Fanuc TP program (LS listing): hosenrohr_ov_h802.ls

/PROG  hosenrohr_ov_h802
/ATTR
COMMENT	= "19-02-26 08:34:14";
PROG_SIZE	= 0;
DEFAULT_GROUP	= 1, 1, *, *, *;
/APPL
    ARC Welding Equipment: 1, *, *, *, *;
/MN
   1:  CALL HOME_ALL;
   1:  UFRAME_NUM = 1;
   1:  UTOOL_NUM = 3;
   1:  COL GUARD ADJUST 150;
   1:  ! -- Layer/Ebene 72 -- !;
   1:  PR[91] = PR[90];
   1:  PR[GP1:91,1] = PR[GP1:90,1] + -1.017;
   1:  PR[GP1:91,2] = PR[GP1:90,2] + 18.874;
   1:  PR[GP1:91,3] = PR[GP1:90,3] + 44.225;
   1:  !Sicherheitspunkt!;
   1:  PR[92] = PR[91];
   1:  PR[92] = PR[GP1:92,3] + 50;
   1:J PR[92];
   1:  !Schweissanfang anfahren!;
   1:L PR[91] R[100]mm/sec CNT100;
   1:  CALL LASER_DRAHT_START;
   1:  PR[GP1:91,1] = PR[GP1:90,1] + -3.858;
   1:  PR[GP1:91,2] = PR[GP1:90,2] + 20.009;
   1:L PR[91] R[100]mm/sec CNT100;
   1:  PR[GP1:91,1] = PR[GP1:90,1] + -5.422;
   1:  PR[GP1:91,2] = PR[GP1:90,2] + 20.569;
   1:L PR[91] R[100]mm/sec CNT100;
   1:  PR[GP1:91,1] = PR[GP1:90,1] + -10.694;
   1:  PR[GP1:91,2] = PR[GP1:90,2] + 21.232;
   1:L PR[91] R[100]mm/sec CNT100;
   1:  PR[GP1:91,1] = PR[GP1:90,1] + -11.339;
   1:  PR[GP1:91,2] = PR[GP1:90,2] + 21.294;
   1:L PR[91] R[100]mm/sec CNT100;
   1:  PR[GP1:91,1] = PR[GP1:90,1] + -17.031;
   1:  PR[GP1:91,2] = PR[GP1:90,2] + 20.547;
   1:L PR[91] R[100]mm/sec CNT100;
   1:  PR[GP1:91,1] = PR[GP1:90,1] + -17.231;
   1:  PR[GP1:91,2] = PR[GP1:90,2] + 20.514;
   1:L PR[91] R[100]mm/sec CNT100;
   1:  PR[GP1:91,1] = PR[GP1:90,1] + -22.722;
   1:  PR[GP1:91,2] = PR[GP1:90,2] + 18.298;
   1:L PR[91] R[100]mm/sec CNT100;
   1:  PR[GP1:91,1] = PR[GP1:90,1] + -27.488;
   1:  PR[GP1:91,2] = PR[GP1:90,2] + 14.829;
   1:L PR[91] R[100]mm/sec CNT100;
   1:  PR[GP1:91,1] = PR[GP1:90,1] + -27.511;
   1:  PR[GP1:91,2] = PR[GP1:90,2] + 14.804;
   1:L PR[91] R[100]mm/sec CNT100;
   1:  PR[GP1:91,1] = PR[GP1:90,1] + -30.986;
   1:  PR[GP1:91,2] = PR[GP1:90,2] + 10.489;
   1:L PR[91] R[100]mm/sec CNT100;
   1:  PR[GP1:91,1] = PR[GP1:90,1] + -31.085;
   1:  PR[GP1:91,2] = PR[GP1:90,2] + 10.338;
   1:L PR[91] R[100]mm/sec CNT100;
   1:  PR[GP1:91,1] = PR[GP1:90,1] + -33.300;
   1:  PR[GP1:91,2] = PR[GP1:90,2] + 5.293;
   1:L PR[91] R[100]mm/sec CNT100;
   1:  PR[GP1:91,1] = PR[GP1:90,1] + -33.354;
   1:  PR[GP1:91,2] = PR[GP1:90,2] + 5.083;
   1:L PR[91] R[100]mm/sec CNT100;
   1:  PR[GP1:91,1] = PR[GP1:90,1] + -33.385;
   1:  PR[GP1:91,2] = PR[GP1:90,2] + 4.702;
   1:L PR[91] R[100]mm/sec CNT100;
   1:  PR[GP1:91,1] = PR[GP1:90,1] + -34.086;
   1:  PR[GP1:91,2] = PR[GP1:90,2] + -0.354;
   1:L PR[91] R[100]mm/sec CNT100;
   1:  PR[GP1:91,1] = PR[GP1:90,1] + -34.060;
   1:  PR[GP1:91,2] = PR[GP1:90,2] + -0.674;
   1:L PR[91] R[100]mm/sec CNT100;
   1:  PR[GP1:91,1] = PR[GP1:90,1] + -33.363;
   1:  PR[GP1:91,2] = PR[GP1:90,2] + -5.673;
   1:L PR[91] R[100]mm/sec CNT100;
   1:  PR[GP1:91,1] = PR[GP1:90,1] + -33.300;
   1:  PR[GP1:91,2] = PR[GP1:90,2] + -5.917;
   1:L PR[91] R[100]mm/sec CNT100;
   1:  PR[GP1:91,1] = PR[GP1:90,1] + -33.156;
   1:  PR[GP1:91,2] = PR[GP1:90,2] + -6.238;
   1:L PR[91] R[100]mm/sec CNT100;
   1:  PR[GP1:91,1] = PR[GP1:90,1] + -31.078;
   1:  PR[GP1:91,2] = PR[GP1:90,2] + -10.975;
   1:L PR[91] R[100]mm/sec CNT100;
   1:  PR[GP1:91,1] = PR[GP1:90,1] + -30.980;
   1:  PR[GP1:91,2] = PR[GP1:90,2] + -11.125;
   1:L PR[91] R[100]mm/sec CNT100;
   1:  PR[GP1:91,1] = PR[GP1:90,1] + -27.495;
   1:  PR[GP1:91,2] = PR[GP1:90,2] + -15.443;
   1:L PR[91] R[100]mm/sec CNT100;
   1:  PR[GP1:91,1] = PR[GP1:90,1] + -27.473;
   1:  PR[GP1:91,2] = PR[GP1:90,2] + -15.467;
   1:L PR[91] R[100]mm/sec CNT100;
   1:  PR[GP1:91,1] = PR[GP1:90,1] + -22.696;
   1:  PR[GP1:91,2] = PR[GP1:90,2] + -18.937;
   1:L PR[91] R[100]mm/sec CNT100;
   1:  PR[GP1:91,1] = PR[GP1:90,1] + -17.195;
   1:  PR[GP1:91,2] = PR[GP1:90,2] + -21.148;
   1:L PR[91] R[100]mm/sec CNT100;
   1:  PR[GP1:91,1] = PR[GP1:90,1] + -16.992;
   1:  PR[GP1:91,2] = PR[GP1:90,2] + -21.180;
   1:L PR[91] R[100]mm/sec CNT100;
   1:  PR[GP1:91,1] = PR[GP1:90,1] + -11.296;
   1:  PR[GP1:91,2] = PR[GP1:90,2] + -21.918;
   1:L PR[91] R[100]mm/sec CNT100;
   1:  PR[GP1:91,1] = PR[GP1:90,1] + -10.640;
   1:  PR[GP1:91,2] = PR[GP1:90,2] + -21.853;
   1:L PR[91] R[100]mm/sec CNT100;
   1:  PR[GP1:91,1] = PR[GP1:90,1] + -5.365;
   1:  PR[GP1:91,2] = PR[GP1:90,2] + -21.179;
   1:L PR[91] R[100]mm/sec CNT100;
   1:  PR[GP1:91,1] = PR[GP1:90,1] + -4.473;
   1:  PR[GP1:91,2] = PR[GP1:90,2] + -20.868;
   1:L PR[91] R[100]mm/sec CNT100;
   1:  PR[GP1:91,1] = PR[GP1:90,1] + -1.022;
   1:  PR[GP1:91,2] = PR[GP1:90,2] + -19.515;
   1:L PR[91] R[100]mm/sec CNT100;
   1:  PR[GP1:91,1] = PR[GP1:90,1] + 0.411;
   1:  PR[GP1:91,2] = PR[GP1:90,2] + -19.282;
   1:L PR[91] R[100]mm/sec CNT100;
   1:  PR[GP1:91,1] = PR[GP1:90,1] + 1.272;
   1:  PR[GP1:91,2] = PR[GP1:90,2] + -19.552;
   1:L PR[91] R[100]mm/sec CNT100;
   1:  PR[GP1:91,1] = PR[GP1:90,1] + 4.630;
   1:  PR[GP1:91,2] = PR[GP1:90,2] + -20.867;
   1:L PR[91] R[100]mm/sec CNT100;
   1:  PR[GP1:91,1] = PR[GP1:90,1] + 5.411;
   1:  PR[GP1:91,2] = PR[GP1:90,2] + -21.143;
   1:L PR[91] R[100]mm/sec CNT100;
   1:  PR[GP1:91,1] = PR[GP1:90,1] + 10.700;
   1:  PR[GP1:91,2] = PR[GP1:90,2] + -21.827;
   1:L PR[91] R[100]mm/sec CNT100;
   1:  PR[GP1:91,1] = PR[GP1:90,1] + 10.853;
   1:  PR[GP1:91,2] = PR[GP1:90,2] + -21.859;
   1:L PR[91] R[100]mm/sec CNT100;
   1:  PR[GP1:91,1] = PR[GP1:90,1] + 11.450;
   1:  PR[GP1:91,2] = PR[GP1:90,2] + -21.918;
   1:L PR[91] R[100]mm/sec CNT100;
   1:  PR[GP1:91,1] = PR[GP1:90,1] + 17.146;
   1:  PR[GP1:91,2] = PR[GP1:90,2] + -21.180;
   1:L PR[91] R[100]mm/sec CNT100;
   1:  PR[GP1:91,1] = PR[GP1:90,1] + 17.349;
   1:  PR[GP1:91,2] = PR[GP1:90,2] + -21.148;
   1:L PR[91] R[100]mm/sec CNT100;
   1:  PR[GP1:91,1] = PR[GP1:90,1] + 22.851;
   1:  PR[GP1:91,2] = PR[GP1:90,2] + -18.939;
   1:L PR[91] R[100]mm/sec CNT100;
   1:  PR[GP1:91,1] = PR[GP1:90,1] + 27.626;
   1:  PR[GP1:91,2] = PR[GP1:90,2] + -15.472;
   1:L PR[91] R[100]mm/sec CNT100;
   1:  PR[GP1:91,1] = PR[GP1:90,1] + 27.648;
   1:  PR[GP1:91,2] = PR[GP1:90,2] + -15.448;
   1:L PR[91] R[100]mm/sec CNT100;
   1:  PR[GP1:91,1] = PR[GP1:90,1] + 31.132;
   1:  PR[GP1:91,2] = PR[GP1:90,2] + -11.122;
   1:L PR[91] R[100]mm/sec CNT100;
   1:  PR[GP1:91,1] = PR[GP1:90,1] + 31.234;
   1:  PR[GP1:91,2] = PR[GP1:90,2] + -10.967;
   1:L PR[91] R[100]mm/sec CNT100;
   1:  PR[GP1:91,1] = PR[GP1:90,1] + 33.454;
   1:  PR[GP1:91,2] = PR[GP1:90,2] + -5.943;
   1:L PR[91] R[100]mm/sec CNT100;
   1:  PR[GP1:91,1] = PR[GP1:90,1] + 33.508;
   1:  PR[GP1:91,2] = PR[GP1:90,2] + -5.738;
   1:L PR[91] R[100]mm/sec CNT100;
   1:  PR[GP1:91,1] = PR[GP1:90,1] + 33.540;
   1:  PR[GP1:91,2] = PR[GP1:90,2] + -5.345;
   1:L PR[91] R[100]mm/sec CNT100;
   1:  PR[GP1:91,1] = PR[GP1:90,1] + 34.242;
   1:  PR[GP1:91,2] = PR[GP1:90,2] + -0.271;
   1:L PR[91] R[100]mm/sec CNT100;
   1:  PR[GP1:91,1] = PR[GP1:90,1] + 34.215;
   1:  PR[GP1:91,2] = PR[GP1:90,2] + 0.065;
   1:L PR[91] R[100]mm/sec CNT100;
   1:  PR[GP1:91,1] = PR[GP1:90,1] + 33.520;
   1:  PR[GP1:91,2] = PR[GP1:90,2] + 5.069;
   1:L PR[91] R[100]mm/sec CNT100;
   1:  PR[GP1:91,1] = PR[GP1:90,1] + 33.456;
   1:  PR[GP1:91,2] = PR[GP1:90,2] + 5.313;
   1:L PR[91] R[100]mm/sec CNT100;
   1:  PR[GP1:91,1] = PR[GP1:90,1] + 31.241;
   1:  PR[GP1:91,2] = PR[GP1:90,2] + 10.332;
   1:L PR[91] R[100]mm/sec CNT100;
   1:  PR[GP1:91,1] = PR[GP1:90,1] + 31.139;
   1:  PR[GP1:91,2] = PR[GP1:90,2] + 10.487;
   1:L PR[91] R[100]mm/sec CNT100;
   1:  PR[GP1:91,1] = PR[GP1:90,1] + 27.664;
   1:  PR[GP1:91,2] = PR[GP1:90,2] + 14.809;
   1:L PR[91] R[100]mm/sec CNT100;
   1:  PR[GP1:91,1] = PR[GP1:90,1] + 27.641;
   1:  PR[GP1:91,2] = PR[GP1:90,2] + 14.834;
   1:L PR[91] R[100]mm/sec CNT100;
   1:  PR[GP1:91,1] = PR[GP1:90,1] + 22.877;
   1:  PR[GP1:91,2] = PR[GP1:90,2] + 18.301;
   1:L PR[91] R[100]mm/sec CNT100;
   1:  PR[GP1:91,1] = PR[GP1:90,1] + 17.385;
   1:  PR[GP1:91,2] = PR[GP1:90,2] + 20.514;
   1:L PR[91] R[100]mm/sec CNT100;
   1:  PR[GP1:91,1] = PR[GP1:90,1] + 17.184;
   1:  PR[GP1:91,2] = PR[GP1:90,2] + 20.547;
   1:L PR[91] R[100]mm/sec CNT100;
   1:  PR[GP1:91,1] = PR[GP1:90,1] + 11.493;
   1:  PR[GP1:91,2] = PR[GP1:90,2] + 21.294;
   1:L PR[91] R[100]mm/sec CNT100;
   1:  PR[GP1:91,1] = PR[GP1:90,1] + 10.848;
   1:  PR[GP1:91,2] = PR[GP1:90,2] + 21.232;
   1:L PR[91] R[100]mm/sec CNT100;
   1:  PR[GP1:91,1] = PR[GP1:90,1] + 5.555;
   1:  PR[GP1:91,2] = PR[GP1:90,2] + 20.565;
   1:L PR[91] R[100]mm/sec CNT100;
   1:  PR[GP1:91,1] = PR[GP1:90,1] + 5.340;
   1:  PR[GP1:91,2] = PR[GP1:90,2] + 20.494;
   1:L PR[91] R[100]mm/sec CNT100;
   1:  PR[GP1:91,1] = PR[GP1:90,1] + 4.017;
   1:  PR[GP1:91,2] = PR[GP1:90,2] + 20.009;
   1:L PR[91] R[100]mm/sec CNT100;
   1:  PR[GP1:91,1] = PR[GP1:90,1] + 1.242;
   1:  PR[GP1:91,2] = PR[GP1:90,2] + 18.902;
   1:L PR[91] R[100]mm/sec CNT100;
   1:  PR[GP1:91,1] = PR[GP1:90,1] + 0.855;
   1:  PR[GP1:91,2] = PR[GP1:90,2] + 18.802;
   1:L PR[91] R[100]mm/sec CNT100;
   1:  PR[GP1:91,1] = PR[GP1:90,1] + 0.519;
   1:  PR[GP1:91,2] = PR[GP1:90,2] + 18.647;
   1:L PR[91] R[100]mm/sec CNT100;
   1:  ! -- Layer/Ebene 73 -- !;
   1:  PR[91] = PR[90];
   1:  PR[GP1:91,1] = PR[GP1:90,1] + -1.002;
   1:  PR[GP1:91,2] = PR[GP1:90,2] + 19.074;
   1:  PR[GP1:91,3] = PR[GP1:90,3] + 44.835;
   1:L PR[91] R[100]mm/sec CNT100;
   1:  PR[GP1:91,1] = PR[GP1:90,1] + -3.287;
   1:  PR[GP1:91,2] = PR[GP1:90,2] + 19.987;
   1:L PR[91] R[100]mm/sec CNT100;
   1:  PR[GP1:91,1] = PR[GP1:90,1] + -5.044;
   1:  PR[GP1:91,2] = PR[GP1:90,2] + 20.628;
   1:L PR[91] R[100]mm/sec CNT100;
   1:  PR[GP1:91,1] = PR[GP1:90,1] + -5.181;
   1:  PR[GP1:91,2] = PR[GP1:90,2] + 20.671;
   1:L PR[91] R[100]mm/sec CNT100;
   1:  PR[GP1:91,1] = PR[GP1:90,1] + -10.231;
   1:  PR[GP1:91,2] = PR[GP1:90,2] + 21.306;
   1:L PR[91] R[100]mm/sec CNT100;
   1:  PR[GP1:91,1] = PR[GP1:90,1] + -11.140;
   1:  PR[GP1:91,2] = PR[GP1:90,2] + 21.393;
   1:L PR[91] R[100]mm/sec CNT100;
   1:  PR[GP1:91,1] = PR[GP1:90,1] + -16.581;
   1:  PR[GP1:91,2] = PR[GP1:90,2] + 20.679;
   1:L PR[91] R[100]mm/sec CNT100;
   1:  PR[GP1:91,1] = PR[GP1:90,1] + -17.045;
   1:  PR[GP1:91,2] = PR[GP1:90,2] + 20.605;
   1:L PR[91] R[100]mm/sec CNT100;
   1:  PR[GP1:91,1] = PR[GP1:90,1] + -22.543;
   1:  PR[GP1:91,2] = PR[GP1:90,2] + 18.372;
   1:L PR[91] R[100]mm/sec CNT100;
   1:  PR[GP1:91,1] = PR[GP1:90,1] + -25.480;
   1:  PR[GP1:91,2] = PR[GP1:90,2] + 16.189;
   1:L PR[91] R[100]mm/sec CNT100;
   1:  PR[GP1:91,1] = PR[GP1:90,1] + -27.252;
   1:  PR[GP1:91,2] = PR[GP1:90,2] + 14.898;
   1:L PR[91] R[100]mm/sec CNT100;
   1:  PR[GP1:91,1] = PR[GP1:90,1] + -30.851;
   1:  PR[GP1:91,2] = PR[GP1:90,2] + 10.438;
   1:L PR[91] R[100]mm/sec CNT100;
   1:  PR[GP1:91,1] = PR[GP1:90,1] + -30.874;
   1:  PR[GP1:91,2] = PR[GP1:90,2] + 10.403;
   1:L PR[91] R[100]mm/sec CNT100;
   1:  PR[GP1:91,1] = PR[GP1:90,1] + -30.924;
   1:  PR[GP1:91,2] = PR[GP1:90,2] + 10.292;
   1:L PR[91] R[100]mm/sec CNT100;
   1:  PR[GP1:91,1] = PR[GP1:90,1] + -33.125;
   1:  PR[GP1:91,2] = PR[GP1:90,2] + 5.268;
   1:L PR[91] R[100]mm/sec CNT100;
   1:  PR[GP1:91,1] = PR[GP1:90,1] + -33.144;
   1:  PR[GP1:91,2] = PR[GP1:90,2] + 5.195;
   1:L PR[91] R[100]mm/sec CNT100;
   1:  PR[GP1:91,1] = PR[GP1:90,1] + -33.163;
   1:  PR[GP1:91,2] = PR[GP1:90,2] + 4.957;
   1:L PR[91] R[100]mm/sec CNT100;
   1:  PR[GP1:91,1] = PR[GP1:90,1] + -33.900;
   1:  PR[GP1:91,2] = PR[GP1:90,2] + -0.354;
   1:L PR[91] R[100]mm/sec CNT100;
   1:  PR[GP1:91,1] = PR[GP1:90,1] + -33.885;
   1:  PR[GP1:91,2] = PR[GP1:90,2] + -0.535;
   1:L PR[91] R[100]mm/sec CNT100;
   1:  PR[GP1:91,1] = PR[GP1:90,1] + -33.153;
   1:  PR[GP1:91,2] = PR[GP1:90,2] + -5.784;
   1:L PR[91] R[100]mm/sec CNT100;
   1:  PR[GP1:91,1] = PR[GP1:90,1] + -33.125;
   1:  PR[GP1:91,2] = PR[GP1:90,2] + -5.892;
   1:L PR[91] R[100]mm/sec CNT100;
   1:  PR[GP1:91,1] = PR[GP1:90,1] + -33.040;
   1:  PR[GP1:91,2] = PR[GP1:90,2] + -6.081;
   1:L PR[91] R[100]mm/sec CNT100;
   1:  PR[GP1:91,1] = PR[GP1:90,1] + -30.863;
   1:  PR[GP1:91,2] = PR[GP1:90,2] + -11.044;
   1:L PR[91] R[100]mm/sec CNT100;
   1:  PR[GP1:91,1] = PR[GP1:90,1] + -30.844;
   1:  PR[GP1:91,2] = PR[GP1:90,2] + -11.074;
   1:L PR[91] R[100]mm/sec CNT100;
   1:  PR[GP1:91,1] = PR[GP1:90,1] + -27.236;
   1:  PR[GP1:91,2] = PR[GP1:90,2] + -15.537;
   1:L PR[91] R[100]mm/sec CNT100;
   1:  PR[GP1:91,1] = PR[GP1:90,1] + -25.483;
   1:  PR[GP1:91,2] = PR[GP1:90,2] + -16.812;
   1:L PR[91] R[100]mm/sec CNT100;
   1:  PR[GP1:91,1] = PR[GP1:90,1] + -22.517;
   1:  PR[GP1:91,2] = PR[GP1:90,2] + -19.010;
   1:L PR[91] R[100]mm/sec CNT100;
   1:  PR[GP1:91,1] = PR[GP1:90,1] + -17.009;
   1:  PR[GP1:91,2] = PR[GP1:90,2] + -21.238;
   1:L PR[91] R[100]mm/sec CNT100;
   1:  PR[GP1:91,1] = PR[GP1:90,1] + -16.542;
   1:  PR[GP1:91,2] = PR[GP1:90,2] + -21.312;
   1:L PR[91] R[100]mm/sec CNT100;
   1:  PR[GP1:91,1] = PR[GP1:90,1] + -11.097;
   1:  PR[GP1:91,2] = PR[GP1:90,2] + -22.018;
   1:L PR[91] R[100]mm/sec CNT100;
   1:  PR[GP1:91,1] = PR[GP1:90,1] + -10.175;
   1:  PR[GP1:91,2] = PR[GP1:90,2] + -21.926;
   1:L PR[91] R[100]mm/sec CNT100;
   1:  PR[GP1:91,1] = PR[GP1:90,1] + -5.149;
   1:  PR[GP1:91,2] = PR[GP1:90,2] + -21.284;
   1:L PR[91] R[100]mm/sec CNT100;
   1:  PR[GP1:91,1] = PR[GP1:90,1] + -4.038;
   1:  PR[GP1:91,2] = PR[GP1:90,2] + -20.897;
   1:L PR[91] R[100]mm/sec CNT100;
   1:  PR[GP1:91,1] = PR[GP1:90,1] + -1.002;
   1:  PR[GP1:91,2] = PR[GP1:90,2] + -19.707;
   1:L PR[91] R[100]mm/sec CNT100;
   1:  PR[GP1:91,1] = PR[GP1:90,1] + 0.577;
   1:  PR[GP1:91,2] = PR[GP1:90,2] + -19.458;
   1:L PR[91] R[100]mm/sec CNT100;
   1:  PR[GP1:91,1] = PR[GP1:90,1] + 0.929;
   1:  PR[GP1:91,2] = PR[GP1:90,2] + -19.646;
   1:L PR[91] R[100]mm/sec CNT100;
   1:  PR[GP1:91,1] = PR[GP1:90,1] + 1.247;
   1:  PR[GP1:91,2] = PR[GP1:90,2] + -19.742;
   1:L PR[91] R[100]mm/sec CNT100;
   1:  PR[GP1:91,1] = PR[GP1:90,1] + 4.196;
   1:  PR[GP1:91,2] = PR[GP1:90,2] + -20.896;
   1:L PR[91] R[100]mm/sec CNT100;
   1:  PR[GP1:91,1] = PR[GP1:90,1] + 5.172;
   1:  PR[GP1:91,2] = PR[GP1:90,2] + -21.240;
   1:L PR[91] R[100]mm/sec CNT100;
   1:  PR[GP1:91,1] = PR[GP1:90,1] + 10.180;
   1:  PR[GP1:91,2] = PR[GP1:90,2] + -21.888;
   1:L PR[91] R[100]mm/sec CNT100;
   1:  PR[GP1:91,1] = PR[GP1:90,1] + 10.388;
   1:  PR[GP1:91,2] = PR[GP1:90,2] + -21.932;
   1:L PR[91] R[100]mm/sec CNT100;
   1:  PR[GP1:91,1] = PR[GP1:90,1] + 11.251;
   1:  PR[GP1:91,2] = PR[GP1:90,2] + -22.018;
   1:L PR[91] R[100]mm/sec CNT100;
   1:  PR[GP1:91,1] = PR[GP1:90,1] + 16.697;
   1:  PR[GP1:91,2] = PR[GP1:90,2] + -21.312;
   1:L PR[91] R[100]mm/sec CNT100;
   1:  PR[GP1:91,1] = PR[GP1:90,1] + 17.164;
   1:  PR[GP1:91,2] = PR[GP1:90,2] + -21.238;
   1:L PR[91] R[100]mm/sec CNT100;
   1:  PR[GP1:91,1] = PR[GP1:90,1] + 22.673;
   1:  PR[GP1:91,2] = PR[GP1:90,2] + -19.012;
   1:L PR[91] R[100]mm/sec CNT100;
   1:  PR[GP1:91,1] = PR[GP1:90,1] + 25.638;
   1:  PR[GP1:91,2] = PR[GP1:90,2] + -16.814;
   1:L PR[91] R[100]mm/sec CNT100;
   1:  PR[GP1:91,1] = PR[GP1:90,1] + 27.390;
   1:  PR[GP1:91,2] = PR[GP1:90,2] + -15.541;
   1:L PR[91] R[100]mm/sec CNT100;
   1:  PR[GP1:91,1] = PR[GP1:90,1] + 30.998;
   1:  PR[GP1:91,2] = PR[GP1:90,2] + -11.069;
   1:L PR[91] R[100]mm/sec CNT100;
   1:  PR[GP1:91,1] = PR[GP1:90,1] + 31.020;
   1:  PR[GP1:91,2] = PR[GP1:90,2] + -11.036;
   1:L PR[91] R[100]mm/sec CNT100;
   1:  PR[GP1:91,1] = PR[GP1:90,1] + 33.280;
   1:  PR[GP1:91,2] = PR[GP1:90,2] + -5.916;
   1:L PR[91] R[100]mm/sec CNT100;
   1:  PR[GP1:91,1] = PR[GP1:90,1] + 33.298;
   1:  PR[GP1:91,2] = PR[GP1:90,2] + -5.846;
   1:L PR[91] R[100]mm/sec CNT100;
   1:  PR[GP1:91,1] = PR[GP1:90,1] + 33.318;
   1:  PR[GP1:91,2] = PR[GP1:90,2] + -5.601;
   1:L PR[91] R[100]mm/sec CNT100;
   1:  PR[GP1:91,1] = PR[GP1:90,1] + 34.056;
   1:  PR[GP1:91,2] = PR[GP1:90,2] + -0.271;
   1:L PR[91] R[100]mm/sec CNT100;
   1:  PR[GP1:91,1] = PR[GP1:90,1] + 34.040;
   1:  PR[GP1:91,2] = PR[GP1:90,2] + -0.079;
   1:L PR[91] R[100]mm/sec CNT100;
   1:  PR[GP1:91,1] = PR[GP1:90,1] + 33.310;
   1:  PR[GP1:91,2] = PR[GP1:90,2] + 5.176;
   1:L PR[91] R[100]mm/sec CNT100;
   1:  PR[GP1:91,1] = PR[GP1:90,1] + 33.282;
   1:  PR[GP1:91,2] = PR[GP1:90,2] + 5.286;
   1:L PR[91] R[100]mm/sec CNT100;
   1:  PR[GP1:91,1] = PR[GP1:90,1] + 31.027;
   1:  PR[GP1:91,2] = PR[GP1:90,2] + 10.400;
   1:L PR[91] R[100]mm/sec CNT100;
   1:  PR[GP1:91,1] = PR[GP1:90,1] + 31.005;
   1:  PR[GP1:91,2] = PR[GP1:90,2] + 10.433;
   1:L PR[91] R[100]mm/sec CNT100;
   1:  PR[GP1:91,1] = PR[GP1:90,1] + 27.406;
   1:  PR[GP1:91,2] = PR[GP1:90,2] + 14.902;
   1:L PR[91] R[100]mm/sec CNT100;
   1:  PR[GP1:91,1] = PR[GP1:90,1] + 25.636;
   1:  PR[GP1:91,2] = PR[GP1:90,2] + 16.190;
   1:L PR[91] R[100]mm/sec CNT100;
   1:  PR[GP1:91,1] = PR[GP1:90,1] + 22.698;
   1:  PR[GP1:91,2] = PR[GP1:90,2] + 18.374;
   1:L PR[91] R[100]mm/sec CNT100;
   1:  PR[GP1:91,1] = PR[GP1:90,1] + 17.199;
   1:  PR[GP1:91,2] = PR[GP1:90,2] + 20.605;
   1:L PR[91] R[100]mm/sec CNT100;
   1:  PR[GP1:91,1] = PR[GP1:90,1] + 16.735;
   1:  PR[GP1:91,2] = PR[GP1:90,2] + 20.679;
   1:L PR[91] R[100]mm/sec CNT100;
   1:  PR[GP1:91,1] = PR[GP1:90,1] + 11.294;
   1:  PR[GP1:91,2] = PR[GP1:90,2] + 21.394;
   1:L PR[91] R[100]mm/sec CNT100;
   1:  PR[GP1:91,1] = PR[GP1:90,1] + 10.386;
   1:  PR[GP1:91,2] = PR[GP1:90,2] + 21.306;
   1:L PR[91] R[100]mm/sec CNT100;
   1:  PR[GP1:91,1] = PR[GP1:90,1] + 5.339;
   1:  PR[GP1:91,2] = PR[GP1:90,2] + 20.670;
   1:L PR[91] R[100]mm/sec CNT100;
   1:  PR[GP1:91,1] = PR[GP1:90,1] + 5.047;
   1:  PR[GP1:91,2] = PR[GP1:90,2] + 20.575;
   1:L PR[91] R[100]mm/sec CNT100;
   1:  PR[GP1:91,1] = PR[GP1:90,1] + 3.442;
   1:  PR[GP1:91,2] = PR[GP1:90,2] + 19.986;
   1:L PR[91] R[100]mm/sec CNT100;
   1:  PR[GP1:91,1] = PR[GP1:90,1] + 1.226;
   1:  PR[GP1:91,2] = PR[GP1:90,2] + 19.101;
   1:L PR[91] R[100]mm/sec CNT100;
   1:  PR[GP1:91,1] = PR[GP1:90,1] + 0.926;
   1:  PR[GP1:91,2] = PR[GP1:90,2] + 19.024;
   1:L PR[91] R[100]mm/sec CNT100;
   1:  PR[GP1:91,1] = PR[GP1:90,1] + 0.534;
   1:  PR[GP1:91,2] = PR[GP1:90,2] + 18.843;
   1:L PR[91] R[100]mm/sec CNT100;
   1:  ! -- Layer/Ebene 74 -- !;
   1:  PR[91] = PR[90];
   1:  PR[GP1:91,1] = PR[GP1:90,1] + -0.986;
   1:  PR[GP1:91,2] = PR[GP1:90,2] + 19.274;
   1:  PR[GP1:91,3] = PR[GP1:90,3] + 45.445;
   1:L PR[91] R[100]mm/sec CNT100;
   1:  PR[GP1:91,1] = PR[GP1:90,1] + -2.711;
   1:  PR[GP1:91,2] = PR[GP1:90,2] + 19.963;
   1:L PR[91] R[100]mm/sec CNT100;
   1:  PR[GP1:91,1] = PR[GP1:90,1] + -4.778;
   1:  PR[GP1:91,2] = PR[GP1:90,2] + 20.717;
   1:L PR[91] R[100]mm/sec CNT100;
   1:  PR[GP1:91,1] = PR[GP1:90,1] + -4.964;
   1:  PR[GP1:91,2] = PR[GP1:90,2] + 20.776;
   1:L PR[91] R[100]mm/sec CNT100;
   1:  PR[GP1:91,1] = PR[GP1:90,1] + -9.769;
   1:  PR[GP1:91,2] = PR[GP1:90,2] + 21.380;
   1:L PR[91] R[100]mm/sec CNT100;
   1:  PR[GP1:91,1] = PR[GP1:90,1] + -10.941;
   1:  PR[GP1:91,2] = PR[GP1:90,2] + 21.493;
   1:L PR[91] R[100]mm/sec CNT100;
   1:  PR[GP1:91,1] = PR[GP1:90,1] + -16.132;
   1:  PR[GP1:91,2] = PR[GP1:90,2] + 20.811;
   1:L PR[91] R[100]mm/sec CNT100;
   1:  PR[GP1:91,1] = PR[GP1:90,1] + -16.861;
   1:  PR[GP1:91,2] = PR[GP1:90,2] + 20.695;
   1:L PR[91] R[100]mm/sec CNT100;
   1:  PR[GP1:91,1] = PR[GP1:90,1] + -22.059;
   1:  PR[GP1:91,2] = PR[GP1:90,2] + 18.590;
   1:L PR[91] R[100]mm/sec CNT100;
   1:  PR[GP1:91,1] = PR[GP1:90,1] + -22.355;
   1:  PR[GP1:91,2] = PR[GP1:90,2] + 18.460;
   1:L PR[91] R[100]mm/sec CNT100;
   1:  PR[GP1:91,1] = PR[GP1:90,1] + -27.062;
   1:  PR[GP1:91,2] = PR[GP1:90,2] + 14.958;
   1:L PR[91] R[100]mm/sec CNT100;
   1:  PR[GP1:91,1] = PR[GP1:90,1] + -28.678;
   1:  PR[GP1:91,2] = PR[GP1:90,2] + 12.917;
   1:L PR[91] R[100]mm/sec CNT100;
   1:  PR[GP1:91,1] = PR[GP1:90,1] + -30.671;
   1:  PR[GP1:91,2] = PR[GP1:90,2] + 10.441;
   1:L PR[91] R[100]mm/sec CNT100;
   1:  PR[GP1:91,1] = PR[GP1:90,1] + -32.946;
   1:  PR[GP1:91,2] = PR[GP1:90,2] + 5.252;
   1:L PR[91] R[100]mm/sec CNT100;
   1:  PR[GP1:91,1] = PR[GP1:90,1] + -33.713;
   1:  PR[GP1:91,2] = PR[GP1:90,2] + -0.353;
   1:L PR[91] R[100]mm/sec CNT100;
   1:  PR[GP1:91,1] = PR[GP1:90,1] + -33.710;
   1:  PR[GP1:91,2] = PR[GP1:90,2] + -0.395;
   1:L PR[91] R[100]mm/sec CNT100;
   1:  PR[GP1:91,1] = PR[GP1:90,1] + -32.945;
   1:  PR[GP1:91,2] = PR[GP1:90,2] + -5.878;
   1:L PR[91] R[100]mm/sec CNT100;
   1:  PR[GP1:91,1] = PR[GP1:90,1] + -32.925;
   1:  PR[GP1:91,2] = PR[GP1:90,2] + -5.924;
   1:L PR[91] R[100]mm/sec CNT100;
   1:  PR[GP1:91,1] = PR[GP1:90,1] + -30.675;
   1:  PR[GP1:91,2] = PR[GP1:90,2] + -11.053;
   1:L PR[91] R[100]mm/sec CNT100;
   1:  PR[GP1:91,1] = PR[GP1:90,1] + -27.048;
   1:  PR[GP1:91,2] = PR[GP1:90,2] + -15.596;
   1:L PR[91] R[100]mm/sec CNT100;
   1:  PR[GP1:91,1] = PR[GP1:90,1] + -22.330;
   1:  PR[GP1:91,2] = PR[GP1:90,2] + -19.099;
   1:L PR[91] R[100]mm/sec CNT100;
   1:  PR[GP1:91,1] = PR[GP1:90,1] + -22.031;
   1:  PR[GP1:91,2] = PR[GP1:90,2] + -19.229;
   1:L PR[91] R[100]mm/sec CNT100;
   1:  PR[GP1:91,1] = PR[GP1:90,1] + -16.825;
   1:  PR[GP1:91,2] = PR[GP1:90,2] + -21.328;
   1:L PR[91] R[100]mm/sec CNT100;
   1:  PR[GP1:91,1] = PR[GP1:90,1] + -16.093;
   1:  PR[GP1:91,2] = PR[GP1:90,2] + -21.444;
   1:L PR[91] R[100]mm/sec CNT100;
   1:  PR[GP1:91,1] = PR[GP1:90,1] + -10.898;
   1:  PR[GP1:91,2] = PR[GP1:90,2] + -22.117;
   1:L PR[91] R[100]mm/sec CNT100;
   1:  PR[GP1:91,1] = PR[GP1:90,1] + -9.710;
   1:  PR[GP1:91,2] = PR[GP1:90,2] + -22.000;
   1:L PR[91] R[100]mm/sec CNT100;
   1:  PR[GP1:91,1] = PR[GP1:90,1] + -4.932;
   1:  PR[GP1:91,2] = PR[GP1:90,2] + -21.389;
   1:L PR[91] R[100]mm/sec CNT100;
   1:  PR[GP1:91,1] = PR[GP1:90,1] + -3.604;
   1:  PR[GP1:91,2] = PR[GP1:90,2] + -20.926;
   1:L PR[91] R[100]mm/sec CNT100;
   1:  PR[GP1:91,1] = PR[GP1:90,1] + -0.982;
   1:  PR[GP1:91,2] = PR[GP1:90,2] + -19.898;
   1:L PR[91] R[100]mm/sec CNT100;
   1:  PR[GP1:91,1] = PR[GP1:90,1] + 0.597;
   1:  PR[GP1:91,2] = PR[GP1:90,2] + -19.657;
   1:L PR[91] R[100]mm/sec CNT100;
   1:  PR[GP1:91,1] = PR[GP1:90,1] + 0.970;
   1:  PR[GP1:91,2] = PR[GP1:90,2] + -19.857;
   1:L PR[91] R[100]mm/sec CNT100;
   1:  PR[GP1:91,1] = PR[GP1:90,1] + 1.231;
   1:  PR[GP1:91,2] = PR[GP1:90,2] + -19.935;
   1:L PR[91] R[100]mm/sec CNT100;
   1:  PR[GP1:91,1] = PR[GP1:90,1] + 3.761;
   1:  PR[GP1:91,2] = PR[GP1:90,2] + -20.926;
   1:L PR[91] R[100]mm/sec CNT100;
   1:  PR[GP1:91,1] = PR[GP1:90,1] + 4.933;
   1:  PR[GP1:91,2] = PR[GP1:90,2] + -21.338;
   1:L PR[91] R[100]mm/sec CNT100;
   1:  PR[GP1:91,1] = PR[GP1:90,1] + 9.660;
   1:  PR[GP1:91,2] = PR[GP1:90,2] + -21.950;
   1:L PR[91] R[100]mm/sec CNT100;
   1:  PR[GP1:91,1] = PR[GP1:90,1] + 9.924;
   1:  PR[GP1:91,2] = PR[GP1:90,2] + -22.006;
   1:L PR[91] R[100]mm/sec CNT100;
   1:  PR[GP1:91,1] = PR[GP1:90,1] + 11.053;
   1:  PR[GP1:91,2] = PR[GP1:90,2] + -22.117;
   1:L PR[91] R[100]mm/sec CNT100;
   1:  PR[GP1:91,1] = PR[GP1:90,1] + 16.248;
   1:  PR[GP1:91,2] = PR[GP1:90,2] + -21.444;
   1:L PR[91] R[100]mm/sec CNT100;
   1:  PR[GP1:91,1] = PR[GP1:90,1] + 16.980;
   1:  PR[GP1:91,2] = PR[GP1:90,2] + -21.328;
   1:L PR[91] R[100]mm/sec CNT100;
   1:  PR[GP1:91,1] = PR[GP1:90,1] + 22.187;
   1:  PR[GP1:91,2] = PR[GP1:90,2] + -19.230;
   1:L PR[91] R[100]mm/sec CNT100;
   1:  PR[GP1:91,1] = PR[GP1:90,1] + 22.485;
   1:  PR[GP1:91,2] = PR[GP1:90,2] + -19.101;
   1:L PR[91] R[100]mm/sec CNT100;
   1:  PR[GP1:91,1] = PR[GP1:90,1] + 27.203;
   1:  PR[GP1:91,2] = PR[GP1:90,2] + -15.598;
   1:L PR[91] R[100]mm/sec CNT100;
   1:  PR[GP1:91,1] = PR[GP1:90,1] + 30.831;
   1:  PR[GP1:91,2] = PR[GP1:90,2] + -11.046;
   1:L PR[91] R[100]mm/sec CNT100;
   1:  PR[GP1:91,1] = PR[GP1:90,1] + 33.101;
   1:  PR[GP1:91,2] = PR[GP1:90,2] + -5.900;
   1:L PR[91] R[100]mm/sec CNT100;
   1:  PR[GP1:91,1] = PR[GP1:90,1] + 33.870;
   1:  PR[GP1:91,2] = PR[GP1:90,2] + -0.273;
   1:L PR[91] R[100]mm/sec CNT100;
   1:  PR[GP1:91,1] = PR[GP1:90,1] + 33.866;
   1:  PR[GP1:91,2] = PR[GP1:90,2] + -0.223;
   1:L PR[91] R[100]mm/sec CNT100;
   1:  PR[GP1:91,1] = PR[GP1:90,1] + 33.103;
   1:  PR[GP1:91,2] = PR[GP1:90,2] + 5.269;
   1:L PR[91] R[100]mm/sec CNT100;
   1:  PR[GP1:91,1] = PR[GP1:90,1] + 30.838;
   1:  PR[GP1:91,2] = PR[GP1:90,2] + 10.410;
   1:L PR[91] R[100]mm/sec CNT100;
   1:  PR[GP1:91,1] = PR[GP1:90,1] + 27.219;
   1:  PR[GP1:91,2] = PR[GP1:90,2] + 14.959;
   1:L PR[91] R[100]mm/sec CNT100;
   1:  PR[GP1:91,1] = PR[GP1:90,1] + 22.510;
   1:  PR[GP1:91,2] = PR[GP1:90,2] + 18.463;
   1:L PR[91] R[100]mm/sec CNT100;
   1:  PR[GP1:91,1] = PR[GP1:90,1] + 22.214;
   1:  PR[GP1:91,2] = PR[GP1:90,2] + 18.592;
   1:L PR[91] R[100]mm/sec CNT100;
   1:  PR[GP1:91,1] = PR[GP1:90,1] + 17.015;
   1:  PR[GP1:91,2] = PR[GP1:90,2] + 20.694;
   1:L PR[91] R[100]mm/sec CNT100;
   1:  PR[GP1:91,1] = PR[GP1:90,1] + 16.286;
   1:  PR[GP1:91,2] = PR[GP1:90,2] + 20.811;
   1:L PR[91] R[100]mm/sec CNT100;
   1:  PR[GP1:91,1] = PR[GP1:90,1] + 11.095;
   1:  PR[GP1:91,2] = PR[GP1:90,2] + 21.493;
   1:L PR[91] R[100]mm/sec CNT100;
   1:  PR[GP1:91,1] = PR[GP1:90,1] + 9.923;
   1:  PR[GP1:91,2] = PR[GP1:90,2] + 21.380;
   1:L PR[91] R[100]mm/sec CNT100;
   1:  PR[GP1:91,1] = PR[GP1:90,1] + 5.122;
   1:  PR[GP1:91,2] = PR[GP1:90,2] + 20.775;
   1:L PR[91] R[100]mm/sec CNT100;
   1:  PR[GP1:91,1] = PR[GP1:90,1] + 4.754;
   1:  PR[GP1:91,2] = PR[GP1:90,2] + 20.655;
   1:L PR[91] R[100]mm/sec CNT100;
   1:  PR[GP1:91,1] = PR[GP1:90,1] + 2.867;
   1:  PR[GP1:91,2] = PR[GP1:90,2] + 19.962;
   1:L PR[91] R[100]mm/sec CNT100;
   1:  PR[GP1:91,1] = PR[GP1:90,1] + 1.209;
   1:  PR[GP1:91,2] = PR[GP1:90,2] + 19.301;
   1:L PR[91] R[100]mm/sec CNT100;
   1:  PR[GP1:91,1] = PR[GP1:90,1] + 0.997;
   1:  PR[GP1:91,2] = PR[GP1:90,2] + 19.246;
   1:L PR[91] R[100]mm/sec CNT100;
   1:  PR[GP1:91,1] = PR[GP1:90,1] + 0.550;
   1:  PR[GP1:91,2] = PR[GP1:90,2] + 19.040;
   1:L PR[91] R[100]mm/sec CNT100;
   1:  ! -- Layer/Ebene 75 -- !;
   1:  PR[91] = PR[90];
   1:  PR[GP1:91,1] = PR[GP1:90,1] + -0.971;
   1:  PR[GP1:91,2] = PR[GP1:90,2] + 19.474;
   1:  PR[GP1:91,3] = PR[GP1:90,3] + 46.055;
   1:L PR[91] R[100]mm/sec CNT100;
   1:  PR[GP1:91,1] = PR[GP1:90,1] + -2.135;
   1:  PR[GP1:91,2] = PR[GP1:90,2] + 19.940;
   1:L PR[91] R[100]mm/sec CNT100;
   1:  PR[GP1:91,1] = PR[GP1:90,1] + -4.511;
   1:  PR[GP1:91,2] = PR[GP1:90,2] + 20.806;
   1:L PR[91] R[100]mm/sec CNT100;
   1:  PR[GP1:91,1] = PR[GP1:90,1] + -4.747;
   1:  PR[GP1:91,2] = PR[GP1:90,2] + 20.881;
   1:L PR[91] R[100]mm/sec CNT100;
   1:  PR[GP1:91,1] = PR[GP1:90,1] + -9.306;
   1:  PR[GP1:91,2] = PR[GP1:90,2] + 21.454;
   1:L PR[91] R[100]mm/sec CNT100;
   1:  PR[GP1:91,1] = PR[GP1:90,1] + -10.742;
   1:  PR[GP1:91,2] = PR[GP1:90,2] + 21.593;
   1:L PR[91] R[100]mm/sec CNT100;
   1:  PR[GP1:91,1] = PR[GP1:90,1] + -15.682;
   1:  PR[GP1:91,2] = PR[GP1:90,2] + 20.944;
   1:L PR[91] R[100]mm/sec CNT100;
   1:  PR[GP1:91,1] = PR[GP1:90,1] + -16.676;
   1:  PR[GP1:91,2] = PR[GP1:90,2] + 20.784;
   1:L PR[91] R[100]mm/sec CNT100;
   1:  PR[GP1:91,1] = PR[GP1:90,1] + -21.635;
   1:  PR[GP1:91,2] = PR[GP1:90,2] + 18.777;
   1:L PR[91] R[100]mm/sec CNT100;
   1:  PR[GP1:91,1] = PR[GP1:90,1] + -22.182;
   1:  PR[GP1:91,2] = PR[GP1:90,2] + 18.538;
   1:L PR[91] R[100]mm/sec CNT100;
   1:  PR[GP1:91,1] = PR[GP1:90,1] + -26.899;
   1:  PR[GP1:91,2] = PR[GP1:90,2] + 15.020;
   1:L PR[91] R[100]mm/sec CNT100;
   1:  PR[GP1:91,1] = PR[GP1:90,1] + -30.490;
   1:  PR[GP1:91,2] = PR[GP1:90,2] + 10.479;
   1:L PR[91] R[100]mm/sec CNT100;
   1:  PR[GP1:91,1] = PR[GP1:90,1] + -32.742;
   1:  PR[GP1:91,2] = PR[GP1:90,2] + 5.296;
   1:L PR[91] R[100]mm/sec CNT100;
   1:  PR[GP1:91,1] = PR[GP1:90,1] + -33.521;
   1:  PR[GP1:91,2] = PR[GP1:90,2] + -0.312;
   1:L PR[91] R[100]mm/sec CNT100;
   1:  PR[GP1:91,1] = PR[GP1:90,1] + -32.746;
   1:  PR[GP1:91,2] = PR[GP1:90,2] + -5.914;
   1:L PR[91] R[100]mm/sec CNT100;
   1:  PR[GP1:91,1] = PR[GP1:90,1] + -30.483;
   1:  PR[GP1:91,2] = PR[GP1:90,2] + -11.116;
   1:L PR[91] R[100]mm/sec CNT100;
   1:  PR[GP1:91,1] = PR[GP1:90,1] + -26.883;
   1:  PR[GP1:91,2] = PR[GP1:90,2] + -15.659;
   1:L PR[91] R[100]mm/sec CNT100;
   1:  PR[GP1:91,1] = PR[GP1:90,1] + -22.157;
   1:  PR[GP1:91,2] = PR[GP1:90,2] + -19.176;
   1:L PR[91] R[100]mm/sec CNT100;
   1:  PR[GP1:91,1] = PR[GP1:90,1] + -21.607;
   1:  PR[GP1:91,2] = PR[GP1:90,2] + -19.415;
   1:L PR[91] R[100]mm/sec CNT100;
   1:  PR[GP1:91,1] = PR[GP1:90,1] + -16.641;
   1:  PR[GP1:91,2] = PR[GP1:90,2] + -21.418;
   1:L PR[91] R[100]mm/sec CNT100;
   1:  PR[GP1:91,1] = PR[GP1:90,1] + -15.644;
   1:  PR[GP1:91,2] = PR[GP1:90,2] + -21.576;
   1:L PR[91] R[100]mm/sec CNT100;
   1:  PR[GP1:91,1] = PR[GP1:90,1] + -10.699;
   1:  PR[GP1:91,2] = PR[GP1:90,2] + -22.217;
   1:L PR[91] R[100]mm/sec CNT100;
   1:  PR[GP1:91,1] = PR[GP1:90,1] + -9.246;
   1:  PR[GP1:91,2] = PR[GP1:90,2] + -22.073;
   1:L PR[91] R[100]mm/sec CNT100;
   1:  PR[GP1:91,1] = PR[GP1:90,1] + -4.716;
   1:  PR[GP1:91,2] = PR[GP1:90,2] + -21.494;
   1:L PR[91] R[100]mm/sec CNT100;
   1:  PR[GP1:91,1] = PR[GP1:90,1] + -3.169;
   1:  PR[GP1:91,2] = PR[GP1:90,2] + -20.955;
   1:L PR[91] R[100]mm/sec CNT100;
   1:  PR[GP1:91,1] = PR[GP1:90,1] + -0.976;
   1:  PR[GP1:91,2] = PR[GP1:90,2] + -20.095;
   1:L PR[91] R[100]mm/sec CNT100;
   1:  PR[GP1:91,1] = PR[GP1:90,1] + -0.287;
   1:  PR[GP1:91,2] = PR[GP1:90,2] + -19.979;
   1:L PR[91] R[100]mm/sec CNT100;
   1:  PR[GP1:91,1] = PR[GP1:90,1] + 0.634;
   1:  PR[GP1:91,2] = PR[GP1:90,2] + -19.864;
   1:L PR[91] R[100]mm/sec CNT100;
   1:  PR[GP1:91,1] = PR[GP1:90,1] + 1.011;
   1:  PR[GP1:91,2] = PR[GP1:90,2] + -20.067;
   1:L PR[91] R[100]mm/sec CNT100;
   1:  PR[GP1:91,1] = PR[GP1:90,1] + 1.215;
   1:  PR[GP1:91,2] = PR[GP1:90,2] + -20.128;
   1:L PR[91] R[100]mm/sec CNT100;
   1:  PR[GP1:91,1] = PR[GP1:90,1] + 3.327;
   1:  PR[GP1:91,2] = PR[GP1:90,2] + -20.955;
   1:L PR[91] R[100]mm/sec CNT100;
   1:  PR[GP1:91,1] = PR[GP1:90,1] + 4.694;
   1:  PR[GP1:91,2] = PR[GP1:90,2] + -21.436;
   1:L PR[91] R[100]mm/sec CNT100;
   1:  PR[GP1:91,1] = PR[GP1:90,1] + 9.140;
   1:  PR[GP1:91,2] = PR[GP1:90,2] + -22.011;
   1:L PR[91] R[100]mm/sec CNT100;
   1:  PR[GP1:91,1] = PR[GP1:90,1] + 9.459;
   1:  PR[GP1:91,2] = PR[GP1:90,2] + -22.079;
   1:L PR[91] R[100]mm/sec CNT100;
   1:  PR[GP1:91,1] = PR[GP1:90,1] + 10.854;
   1:  PR[GP1:91,2] = PR[GP1:90,2] + -22.217;
   1:L PR[91] R[100]mm/sec CNT100;
   1:  PR[GP1:91,1] = PR[GP1:90,1] + 15.799;
   1:  PR[GP1:91,2] = PR[GP1:90,2] + -21.576;
   1:L PR[91] R[100]mm/sec CNT100;
   1:  PR[GP1:91,1] = PR[GP1:90,1] + 16.796;
   1:  PR[GP1:91,2] = PR[GP1:90,2] + -21.417;
   1:L PR[91] R[100]mm/sec CNT100;
   1:  PR[GP1:91,1] = PR[GP1:90,1] + 21.763;
   1:  PR[GP1:91,2] = PR[GP1:90,2] + -19.417;
   1:L PR[91] R[100]mm/sec CNT100;
   1:  PR[GP1:91,1] = PR[GP1:90,1] + 22.312;
   1:  PR[GP1:91,2] = PR[GP1:90,2] + -19.178;
   1:L PR[91] R[100]mm/sec CNT100;
   1:  PR[GP1:91,1] = PR[GP1:90,1] + 27.038;
   1:  PR[GP1:91,2] = PR[GP1:90,2] + -15.661;
   1:L PR[91] R[100]mm/sec CNT100;
   1:  PR[GP1:91,1] = PR[GP1:90,1] + 30.639;
   1:  PR[GP1:91,2] = PR[GP1:90,2] + -11.108;
   1:L PR[91] R[100]mm/sec CNT100;
   1:  PR[GP1:91,1] = PR[GP1:90,1] + 32.896;
   1:  PR[GP1:91,2] = PR[GP1:90,2] + -5.943;
   1:L PR[91] R[100]mm/sec CNT100;
   1:  PR[GP1:91,1] = PR[GP1:90,1] + 33.681;
   1:  PR[GP1:91,2] = PR[GP1:90,2] + -0.291;
   1:L PR[91] R[100]mm/sec CNT100;
   1:  PR[GP1:91,1] = PR[GP1:90,1] + 32.899;
   1:  PR[GP1:91,2] = PR[GP1:90,2] + 5.312;
   1:L PR[91] R[100]mm/sec CNT100;
   1:  PR[GP1:91,1] = PR[GP1:90,1] + 30.647;
   1:  PR[GP1:91,2] = PR[GP1:90,2] + 10.472;
   1:L PR[91] R[100]mm/sec CNT100;
   1:  PR[GP1:91,1] = PR[GP1:90,1] + 27.054;
   1:  PR[GP1:91,2] = PR[GP1:90,2] + 15.022;
   1:L PR[91] R[100]mm/sec CNT100;
   1:  PR[GP1:91,1] = PR[GP1:90,1] + 22.338;
   1:  PR[GP1:91,2] = PR[GP1:90,2] + 18.540;
   1:L PR[91] R[100]mm/sec CNT100;
   1:  PR[GP1:91,1] = PR[GP1:90,1] + 21.790;
   1:  PR[GP1:91,2] = PR[GP1:90,2] + 18.779;
   1:L PR[91] R[100]mm/sec CNT100;
   1:  PR[GP1:91,1] = PR[GP1:90,1] + 16.831;
   1:  PR[GP1:91,2] = PR[GP1:90,2] + 20.784;
   1:L PR[91] R[100]mm/sec CNT100;
   1:  PR[GP1:91,1] = PR[GP1:90,1] + 15.836;
   1:  PR[GP1:91,2] = PR[GP1:90,2] + 20.944;
   1:L PR[91] R[100]mm/sec CNT100;
   1:  PR[GP1:91,1] = PR[GP1:90,1] + 10.896;
   1:  PR[GP1:91,2] = PR[GP1:90,2] + 21.593;
   1:L PR[91] R[100]mm/sec CNT100;
   1:  PR[GP1:91,1] = PR[GP1:90,1] + 9.460;
   1:  PR[GP1:91,2] = PR[GP1:90,2] + 21.454;
   1:L PR[91] R[100]mm/sec CNT100;
   1:  PR[GP1:91,1] = PR[GP1:90,1] + 4.906;
   1:  PR[GP1:91,2] = PR[GP1:90,2] + 20.880;
   1:L PR[91] R[100]mm/sec CNT100;
   1:  PR[GP1:91,1] = PR[GP1:90,1] + 4.461;
   1:  PR[GP1:91,2] = PR[GP1:90,2] + 20.735;
   1:L PR[91] R[100]mm/sec CNT100;
   1:  PR[GP1:91,1] = PR[GP1:90,1] + 2.292;
   1:  PR[GP1:91,2] = PR[GP1:90,2] + 19.939;
   1:L PR[91] R[100]mm/sec CNT100;
   1:  PR[GP1:91,1] = PR[GP1:90,1] + 1.193;
   1:  PR[GP1:91,2] = PR[GP1:90,2] + 19.500;
   1:L PR[91] R[100]mm/sec CNT100;
   1:  PR[GP1:91,1] = PR[GP1:90,1] + 1.069;
   1:  PR[GP1:91,2] = PR[GP1:90,2] + 19.468;
   1:L PR[91] R[100]mm/sec CNT100;
   1:  PR[GP1:91,1] = PR[GP1:90,1] + 0.566;
   1:  PR[GP1:91,2] = PR[GP1:90,2] + 19.236;
   1:L PR[91] R[100]mm/sec CNT100;
   1:  ! -- Layer/Ebene 76 -- !;
   1:  PR[91] = PR[90];
   1:  PR[GP1:91,1] = PR[GP1:90,1] + -0.956;
   1:  PR[GP1:91,2] = PR[GP1:90,2] + 19.675;
   1:  PR[GP1:91,3] = PR[GP1:90,3] + 46.665;
   1:L PR[91] R[100]mm/sec CNT100;
   1:  PR[GP1:91,1] = PR[GP1:90,1] + -1.560;
   1:  PR[GP1:91,2] = PR[GP1:90,2] + 19.916;
   1:L PR[91] R[100]mm/sec CNT100;
   1:  PR[GP1:91,1] = PR[GP1:90,1] + -4.244;
   1:  PR[GP1:91,2] = PR[GP1:90,2] + 20.895;
   1:L PR[91] R[100]mm/sec CNT100;
   1:  PR[GP1:91,1] = PR[GP1:90,1] + -4.531;
   1:  PR[GP1:91,2] = PR[GP1:90,2] + 20.986;
   1:L PR[91] R[100]mm/sec CNT100;
   1:  PR[GP1:91,1] = PR[GP1:90,1] + -8.843;
   1:  PR[GP1:91,2] = PR[GP1:90,2] + 21.528;
   1:L PR[91] R[100]mm/sec CNT100;
   1:  PR[GP1:91,1] = PR[GP1:90,1] + -10.543;
   1:  PR[GP1:91,2] = PR[GP1:90,2] + 21.692;
   1:L PR[91] R[100]mm/sec CNT100;
   1:  PR[GP1:91,1] = PR[GP1:90,1] + -15.233;
   1:  PR[GP1:91,2] = PR[GP1:90,2] + 21.076;
   1:L PR[91] R[100]mm/sec CNT100;
   1:  PR[GP1:91,1] = PR[GP1:90,1] + -16.492;
   1:  PR[GP1:91,2] = PR[GP1:90,2] + 20.874;
   1:L PR[91] R[100]mm/sec CNT100;
   1:  PR[GP1:91,1] = PR[GP1:90,1] + -21.210;
   1:  PR[GP1:91,2] = PR[GP1:90,2] + 18.964;
   1:L PR[91] R[100]mm/sec CNT100;
   1:  PR[GP1:91,1] = PR[GP1:90,1] + -22.011;
   1:  PR[GP1:91,2] = PR[GP1:90,2] + 18.614;
   1:L PR[91] R[100]mm/sec CNT100;
   1:  PR[GP1:91,1] = PR[GP1:90,1] + -26.329;
   1:  PR[GP1:91,2] = PR[GP1:90,2] + 15.405;
   1:L PR[91] R[100]mm/sec CNT100;
   1:  PR[GP1:91,1] = PR[GP1:90,1] + -26.725;
   1:  PR[GP1:91,2] = PR[GP1:90,2] + 15.095;
   1:L PR[91] R[100]mm/sec CNT100;
   1:  PR[GP1:91,1] = PR[GP1:90,1] + -30.334;
   1:  PR[GP1:91,2] = PR[GP1:90,2] + 10.524;
   1:L PR[91] R[100]mm/sec CNT100;
   1:  PR[GP1:91,1] = PR[GP1:90,1] + -32.584;
   1:  PR[GP1:91,2] = PR[GP1:90,2] + 5.310;
   1:L PR[91] R[100]mm/sec CNT100;
   1:  PR[GP1:91,1] = PR[GP1:90,1] + -33.343;
   1:  PR[GP1:91,2] = PR[GP1:90,2] + -0.312;
   1:L PR[91] R[100]mm/sec CNT100;
   1:  PR[GP1:91,1] = PR[GP1:90,1] + -32.583;
   1:  PR[GP1:91,2] = PR[GP1:90,2] + -5.931;
   1:L PR[91] R[100]mm/sec CNT100;
   1:  PR[GP1:91,1] = PR[GP1:90,1] + -32.581;
   1:  PR[GP1:91,2] = PR[GP1:90,2] + -5.943;
   1:L PR[91] R[100]mm/sec CNT100;
   1:  PR[GP1:91,1] = PR[GP1:90,1] + -30.326;
   1:  PR[GP1:91,2] = PR[GP1:90,2] + -11.160;
   1:L PR[91] R[100]mm/sec CNT100;
   1:  PR[GP1:91,1] = PR[GP1:90,1] + -26.709;
   1:  PR[GP1:91,2] = PR[GP1:90,2] + -15.734;
   1:L PR[91] R[100]mm/sec CNT100;
   1:  PR[GP1:91,1] = PR[GP1:90,1] + -26.312;
   1:  PR[GP1:91,2] = PR[GP1:90,2] + -16.044;
   1:L PR[91] R[100]mm/sec CNT100;
   1:  PR[GP1:91,1] = PR[GP1:90,1] + -21.986;
   1:  PR[GP1:91,2] = PR[GP1:90,2] + -19.252;
   1:L PR[91] R[100]mm/sec CNT100;
   1:  PR[GP1:91,1] = PR[GP1:90,1] + -21.182;
   1:  PR[GP1:91,2] = PR[GP1:90,2] + -19.602;
   1:L PR[91] R[100]mm/sec CNT100;
   1:  PR[GP1:91,1] = PR[GP1:90,1] + -16.457;
   1:  PR[GP1:91,2] = PR[GP1:90,2] + -21.508;
   1:L PR[91] R[100]mm/sec CNT100;
   1:  PR[GP1:91,1] = PR[GP1:90,1] + -15.195;
   1:  PR[GP1:91,2] = PR[GP1:90,2] + -21.708;
   1:L PR[91] R[100]mm/sec CNT100;
   1:  PR[GP1:91,1] = PR[GP1:90,1] + -10.500;
   1:  PR[GP1:91,2] = PR[GP1:90,2] + -22.316;
   1:L PR[91] R[100]mm/sec CNT100;
   1:  PR[GP1:91,1] = PR[GP1:90,1] + -8.781;
   1:  PR[GP1:91,2] = PR[GP1:90,2] + -22.146;
   1:L PR[91] R[100]mm/sec CNT100;
   1:  PR[GP1:91,1] = PR[GP1:90,1] + -4.499;
   1:  PR[GP1:91,2] = PR[GP1:90,2] + -21.599;
   1:L PR[91] R[100]mm/sec CNT100;
   1:  PR[GP1:91,1] = PR[GP1:90,1] + -2.734;
   1:  PR[GP1:91,2] = PR[GP1:90,2] + -20.984;
   1:L PR[91] R[100]mm/sec CNT100;
   1:  PR[GP1:91,1] = PR[GP1:90,1] + -0.943;
   1:  PR[GP1:91,2] = PR[GP1:90,2] + -20.282;
   1:L PR[91] R[100]mm/sec CNT100;
   1:  PR[GP1:91,1] = PR[GP1:90,1] + 0.639;
   1:  PR[GP1:91,2] = PR[GP1:90,2] + -20.055;
   1:L PR[91] R[100]mm/sec CNT100;
   1:  PR[GP1:91,1] = PR[GP1:90,1] + 1.053;
   1:  PR[GP1:91,2] = PR[GP1:90,2] + -20.277;
   1:L PR[91] R[100]mm/sec CNT100;
   1:  PR[GP1:91,1] = PR[GP1:90,1] + 1.199;
   1:  PR[GP1:91,2] = PR[GP1:90,2] + -20.321;
   1:L PR[91] R[100]mm/sec CNT100;
   1:  PR[GP1:91,1] = PR[GP1:90,1] + 2.893;
   1:  PR[GP1:91,2] = PR[GP1:90,2] + -20.984;
   1:L PR[91] R[100]mm/sec CNT100;
   1:  PR[GP1:91,1] = PR[GP1:90,1] + 4.455;
   1:  PR[GP1:91,2] = PR[GP1:90,2] + -21.534;
   1:L PR[91] R[100]mm/sec CNT100;
   1:  PR[GP1:91,1] = PR[GP1:90,1] + 8.620;
   1:  PR[GP1:91,2] = PR[GP1:90,2] + -22.073;
   1:L PR[91] R[100]mm/sec CNT100;
   1:  PR[GP1:91,1] = PR[GP1:90,1] + 8.995;
   1:  PR[GP1:91,2] = PR[GP1:90,2] + -22.152;
   1:L PR[91] R[100]mm/sec CNT100;
   1:  PR[GP1:91,1] = PR[GP1:90,1] + 10.655;
   1:  PR[GP1:91,2] = PR[GP1:90,2] + -22.317;
   1:L PR[91] R[100]mm/sec CNT100;
   1:  PR[GP1:91,1] = PR[GP1:90,1] + 15.350;
   1:  PR[GP1:91,2] = PR[GP1:90,2] + -21.708;
   1:L PR[91] R[100]mm/sec CNT100;
   1:  PR[GP1:91,1] = PR[GP1:90,1] + 16.612;
   1:  PR[GP1:91,2] = PR[GP1:90,2] + -21.507;
   1:L PR[91] R[100]mm/sec CNT100;
   1:  PR[GP1:91,1] = PR[GP1:90,1] + 21.338;
   1:  PR[GP1:91,2] = PR[GP1:90,2] + -19.604;
   1:L PR[91] R[100]mm/sec CNT100;
   1:  PR[GP1:91,1] = PR[GP1:90,1] + 22.142;
   1:  PR[GP1:91,2] = PR[GP1:90,2] + -19.254;
   1:L PR[91] R[100]mm/sec CNT100;
   1:  PR[GP1:91,1] = PR[GP1:90,1] + 26.468;
   1:  PR[GP1:91,2] = PR[GP1:90,2] + -16.046;
   1:L PR[91] R[100]mm/sec CNT100;
   1:  PR[GP1:91,1] = PR[GP1:90,1] + 26.865;
   1:  PR[GP1:91,2] = PR[GP1:90,2] + -15.736;
   1:L PR[91] R[100]mm/sec CNT100;
   1:  PR[GP1:91,1] = PR[GP1:90,1] + 30.483;
   1:  PR[GP1:91,2] = PR[GP1:90,2] + -11.153;
   1:L PR[91] R[100]mm/sec CNT100;
   1:  PR[GP1:91,1] = PR[GP1:90,1] + 32.732;
   1:  PR[GP1:91,2] = PR[GP1:90,2] + -5.982;
   1:L PR[91] R[100]mm/sec CNT100;
   1:  PR[GP1:91,1] = PR[GP1:90,1] + 32.737;
   1:  PR[GP1:91,2] = PR[GP1:90,2] + -5.968;
   1:L PR[91] R[100]mm/sec CNT100;
   1:  PR[GP1:91,1] = PR[GP1:90,1] + 33.500;
   1:  PR[GP1:91,2] = PR[GP1:90,2] + -0.312;
   1:L PR[91] R[100]mm/sec CNT100;
   1:  PR[GP1:91,1] = PR[GP1:90,1] + 32.741;
   1:  PR[GP1:91,2] = PR[GP1:90,2] + 5.326;
   1:L PR[91] R[100]mm/sec CNT100;
   1:  PR[GP1:91,1] = PR[GP1:90,1] + 30.490;
   1:  PR[GP1:91,2] = PR[GP1:90,2] + 10.517;
   1:L PR[91] R[100]mm/sec CNT100;
   1:  PR[GP1:91,1] = PR[GP1:90,1] + 26.880;
   1:  PR[GP1:91,2] = PR[GP1:90,2] + 15.097;
   1:L PR[91] R[100]mm/sec CNT100;
   1:  PR[GP1:91,1] = PR[GP1:90,1] + 26.485;
   1:  PR[GP1:91,2] = PR[GP1:90,2] + 15.407;
   1:L PR[91] R[100]mm/sec CNT100;
   1:  PR[GP1:91,1] = PR[GP1:90,1] + 22.167;
   1:  PR[GP1:91,2] = PR[GP1:90,2] + 18.616;
   1:L PR[91] R[100]mm/sec CNT100;
   1:  PR[GP1:91,1] = PR[GP1:90,1] + 21.366;
   1:  PR[GP1:91,2] = PR[GP1:90,2] + 18.966;
   1:L PR[91] R[100]mm/sec CNT100;
   1:  PR[GP1:91,1] = PR[GP1:90,1] + 16.646;
   1:  PR[GP1:91,2] = PR[GP1:90,2] + 20.874;
   1:L PR[91] R[100]mm/sec CNT100;
   1:  PR[GP1:91,1] = PR[GP1:90,1] + 15.387;
   1:  PR[GP1:91,2] = PR[GP1:90,2] + 21.076;
   1:L PR[91] R[100]mm/sec CNT100;
   1:  PR[GP1:91,1] = PR[GP1:90,1] + 10.697;
   1:  PR[GP1:91,2] = PR[GP1:90,2] + 21.692;
   1:L PR[91] R[100]mm/sec CNT100;
   1:  PR[GP1:91,1] = PR[GP1:90,1] + 8.998;
   1:  PR[GP1:91,2] = PR[GP1:90,2] + 21.528;
   1:L PR[91] R[100]mm/sec CNT100;
   1:  PR[GP1:91,1] = PR[GP1:90,1] + 4.689;
   1:  PR[GP1:91,2] = PR[GP1:90,2] + 20.985;
   1:L PR[91] R[100]mm/sec CNT100;
   1:  PR[GP1:91,1] = PR[GP1:90,1] + 4.168;
   1:  PR[GP1:91,2] = PR[GP1:90,2] + 20.815;
   1:L PR[91] R[100]mm/sec CNT100;
   1:  PR[GP1:91,1] = PR[GP1:90,1] + 1.706;
   1:  PR[GP1:91,2] = PR[GP1:90,2] + 19.911;
   1:L PR[91] R[100]mm/sec CNT100;
   1:  PR[GP1:91,1] = PR[GP1:90,1] + 1.213;
   1:  PR[GP1:91,2] = PR[GP1:90,2] + 19.724;
   1:L PR[91] R[100]mm/sec CNT100;
   1:  PR[GP1:91,1] = PR[GP1:90,1] + 0.581;
   1:  PR[GP1:91,2] = PR[GP1:90,2] + 19.433;
   1:L PR[91] R[100]mm/sec CNT100;
   1:  ! -- Layer/Ebene 77 -- !;
   1:  PR[91] = PR[90];
   1:  PR[GP1:91,1] = PR[GP1:90,1] + -0.917;
   1:  PR[GP1:91,2] = PR[GP1:90,2] + 19.868;
   1:  PR[GP1:91,3] = PR[GP1:90,3] + 47.275;
   1:L PR[91] R[100]mm/sec CNT100;
   1:  PR[GP1:91,1] = PR[GP1:90,1] + -3.978;
   1:  PR[GP1:91,2] = PR[GP1:90,2] + 20.984;
   1:L PR[91] R[100]mm/sec CNT100;
   1:  PR[GP1:91,1] = PR[GP1:90,1] + -4.314;
   1:  PR[GP1:91,2] = PR[GP1:90,2] + 21.091;
   1:L PR[91] R[100]mm/sec CNT100;
   1:  PR[GP1:91,1] = PR[GP1:90,1] + -8.380;
   1:  PR[GP1:91,2] = PR[GP1:90,2] + 21.602;
   1:L PR[91] R[100]mm/sec CNT100;
   1:  PR[GP1:91,1] = PR[GP1:90,1] + -10.343;
   1:  PR[GP1:91,2] = PR[GP1:90,2] + 21.792;
   1:L PR[91] R[100]mm/sec CNT100;
   1:  PR[GP1:91,1] = PR[GP1:90,1] + -14.783;
   1:  PR[GP1:91,2] = PR[GP1:90,2] + 21.209;
   1:L PR[91] R[100]mm/sec CNT100;
   1:  PR[GP1:91,1] = PR[GP1:90,1] + -16.307;
   1:  PR[GP1:91,2] = PR[GP1:90,2] + 20.964;
   1:L PR[91] R[100]mm/sec CNT100;
   1:  PR[GP1:91,1] = PR[GP1:90,1] + -20.786;
   1:  PR[GP1:91,2] = PR[GP1:90,2] + 19.151;
   1:L PR[91] R[100]mm/sec CNT100;
   1:  PR[GP1:91,1] = PR[GP1:90,1] + -21.839;
   1:  PR[GP1:91,2] = PR[GP1:90,2] + 18.691;
   1:L PR[91] R[100]mm/sec CNT100;
   1:  PR[GP1:91,1] = PR[GP1:90,1] + -25.947;
   1:  PR[GP1:91,2] = PR[GP1:90,2] + 15.638;
   1:L PR[91] R[100]mm/sec CNT100;
   1:  PR[GP1:91,1] = PR[GP1:90,1] + -26.564;
   1:  PR[GP1:91,2] = PR[GP1:90,2] + 15.155;
   1:L PR[91] R[100]mm/sec CNT100;
   1:  PR[GP1:91,1] = PR[GP1:90,1] + -29.874;
   1:  PR[GP1:91,2] = PR[GP1:90,2] + 10.973;
   1:L PR[91] R[100]mm/sec CNT100;
   1:  PR[GP1:91,1] = PR[GP1:90,1] + -30.173;
   1:  PR[GP1:91,2] = PR[GP1:90,2] + 10.579;
   1:L PR[91] R[100]mm/sec CNT100;
   1:  PR[GP1:91,1] = PR[GP1:90,1] + -32.434;
   1:  PR[GP1:91,2] = PR[GP1:90,2] + 5.332;
   1:L PR[91] R[100]mm/sec CNT100;
   1:  PR[GP1:91,1] = PR[GP1:90,1] + -33.173;
   1:  PR[GP1:91,2] = PR[GP1:90,2] + -0.120;
   1:L PR[91] R[100]mm/sec CNT100;
   1:  PR[GP1:91,1] = PR[GP1:90,1] + -33.189;
   1:  PR[GP1:91,2] = PR[GP1:90,2] + -0.285;
   1:L PR[91] R[100]mm/sec CNT100;
   1:  PR[GP1:91,1] = PR[GP1:90,1] + -32.502;
   1:  PR[GP1:91,2] = PR[GP1:90,2] + -5.316;
   1:L PR[91] R[100]mm/sec CNT100;
   1:  PR[GP1:91,1] = PR[GP1:90,1] + -32.465;
   1:  PR[GP1:91,2] = PR[GP1:90,2] + -5.708;
   1:L PR[91] R[100]mm/sec CNT100;
   1:  PR[GP1:91,1] = PR[GP1:90,1] + -32.431;
   1:  PR[GP1:91,2] = PR[GP1:90,2] + -5.965;
   1:L PR[91] R[100]mm/sec CNT100;
   1:  PR[GP1:91,1] = PR[GP1:90,1] + -30.166;
   1:  PR[GP1:91,2] = PR[GP1:90,2] + -11.215;
   1:L PR[91] R[100]mm/sec CNT100;
   1:  PR[GP1:91,1] = PR[GP1:90,1] + -29.866;
   1:  PR[GP1:91,2] = PR[GP1:90,2] + -11.610;
   1:L PR[91] R[100]mm/sec CNT100;
   1:  PR[GP1:91,1] = PR[GP1:90,1] + -26.548;
   1:  PR[GP1:91,2] = PR[GP1:90,2] + -15.794;
   1:L PR[91] R[100]mm/sec CNT100;
   1:  PR[GP1:91,1] = PR[GP1:90,1] + -25.930;
   1:  PR[GP1:91,2] = PR[GP1:90,2] + -16.278;
   1:L PR[91] R[100]mm/sec CNT100;
   1:  PR[GP1:91,1] = PR[GP1:90,1] + -21.814;
   1:  PR[GP1:91,2] = PR[GP1:90,2] + -19.329;
   1:L PR[91] R[100]mm/sec CNT100;
   1:  PR[GP1:91,1] = PR[GP1:90,1] + -20.758;
   1:  PR[GP1:91,2] = PR[GP1:90,2] + -19.789;
   1:L PR[91] R[100]mm/sec CNT100;
   1:  PR[GP1:91,1] = PR[GP1:90,1] + -16.272;
   1:  PR[GP1:91,2] = PR[GP1:90,2] + -21.598;
   1:L PR[91] R[100]mm/sec CNT100;
   1:  PR[GP1:91,1] = PR[GP1:90,1] + -14.745;
   1:  PR[GP1:91,2] = PR[GP1:90,2] + -21.840;
   1:L PR[91] R[100]mm/sec CNT100;
   1:  PR[GP1:91,1] = PR[GP1:90,1] + -10.302;
   1:  PR[GP1:91,2] = PR[GP1:90,2] + -22.416;
   1:L PR[91] R[100]mm/sec CNT100;
   1:  PR[GP1:91,1] = PR[GP1:90,1] + -8.316;
   1:  PR[GP1:91,2] = PR[GP1:90,2] + -22.220;
   1:L PR[91] R[100]mm/sec CNT100;
   1:  PR[GP1:91,1] = PR[GP1:90,1] + -4.283;
   1:  PR[GP1:91,2] = PR[GP1:90,2] + -21.704;
   1:L PR[91] R[100]mm/sec CNT100;
   1:  PR[GP1:91,1] = PR[GP1:90,1] + -2.299;
   1:  PR[GP1:91,2] = PR[GP1:90,2] + -21.013;
   1:L PR[91] R[100]mm/sec CNT100;
   1:  PR[GP1:91,1] = PR[GP1:90,1] + -0.923;
   1:  PR[GP1:91,2] = PR[GP1:90,2] + -20.474;
   1:L PR[91] R[100]mm/sec CNT100;
   1:  PR[GP1:91,1] = PR[GP1:90,1] + 0.659;
   1:  PR[GP1:91,2] = PR[GP1:90,2] + -20.254;
   1:L PR[91] R[100]mm/sec CNT100;
   1:  PR[GP1:91,1] = PR[GP1:90,1] + 1.094;
   1:  PR[GP1:91,2] = PR[GP1:90,2] + -20.487;
   1:L PR[91] R[100]mm/sec CNT100;
   1:  PR[GP1:91,1] = PR[GP1:90,1] + 1.183;
   1:  PR[GP1:91,2] = PR[GP1:90,2] + -20.514;
   1:L PR[91] R[100]mm/sec CNT100;
   1:  PR[GP1:91,1] = PR[GP1:90,1] + 2.458;
   1:  PR[GP1:91,2] = PR[GP1:90,2] + -21.013;
   1:L PR[91] R[100]mm/sec CNT100;
   1:  PR[GP1:91,1] = PR[GP1:90,1] + 4.216;
   1:  PR[GP1:91,2] = PR[GP1:90,2] + -21.632;
   1:L PR[91] R[100]mm/sec CNT100;
   1:  PR[GP1:91,1] = PR[GP1:90,1] + 8.100;
   1:  PR[GP1:91,2] = PR[GP1:90,2] + -22.135;
   1:L PR[91] R[100]mm/sec CNT100;
   1:  PR[GP1:91,1] = PR[GP1:90,1] + 8.530;
   1:  PR[GP1:91,2] = PR[GP1:90,2] + -22.226;
   1:L PR[91] R[100]mm/sec CNT100;
   1:  PR[GP1:91,1] = PR[GP1:90,1] + 10.457;
   1:  PR[GP1:91,2] = PR[GP1:90,2] + -22.416;
   1:L PR[91] R[100]mm/sec CNT100;
   1:  PR[GP1:91,1] = PR[GP1:90,1] + 14.900;
   1:  PR[GP1:91,2] = PR[GP1:90,2] + -21.840;
   1:L PR[91] R[100]mm/sec CNT100;
   1:  PR[GP1:91,1] = PR[GP1:90,1] + 16.428;
   1:  PR[GP1:91,2] = PR[GP1:90,2] + -21.597;
   1:L PR[91] R[100]mm/sec CNT100;
   1:  PR[GP1:91,1] = PR[GP1:90,1] + 20.914;
   1:  PR[GP1:91,2] = PR[GP1:90,2] + -19.790;
   1:L PR[91] R[100]mm/sec CNT100;
   1:  PR[GP1:91,1] = PR[GP1:90,1] + 21.970;
   1:  PR[GP1:91,2] = PR[GP1:90,2] + -19.331;
   1:L PR[91] R[100]mm/sec CNT100;
   1:  PR[GP1:91,1] = PR[GP1:90,1] + 26.086;
   1:  PR[GP1:91,2] = PR[GP1:90,2] + -16.279;
   1:L PR[91] R[100]mm/sec CNT100;
   1:  PR[GP1:91,1] = PR[GP1:90,1] + 26.703;
   1:  PR[GP1:91,2] = PR[GP1:90,2] + -15.796;
   1:L PR[91] R[100]mm/sec CNT100;
   1:  PR[GP1:91,1] = PR[GP1:90,1] + 30.021;
   1:  PR[GP1:91,2] = PR[GP1:90,2] + -11.604;
   1:L PR[91] R[100]mm/sec CNT100;
   1:  PR[GP1:91,1] = PR[GP1:90,1] + 30.323;
   1:  PR[GP1:91,2] = PR[GP1:90,2] + -11.207;
   1:L PR[91] R[100]mm/sec CNT100;
   1:  PR[GP1:91,1] = PR[GP1:90,1] + 32.473;
   1:  PR[GP1:91,2] = PR[GP1:90,2] + -6.263;
   1:L PR[91] R[100]mm/sec CNT100;
   1:  PR[GP1:91,1] = PR[GP1:90,1] + 32.587;
   1:  PR[GP1:91,2] = PR[GP1:90,2] + -5.989;
   1:L PR[91] R[100]mm/sec CNT100;
   1:  PR[GP1:91,1] = PR[GP1:90,1] + 33.329;
   1:  PR[GP1:91,2] = PR[GP1:90,2] + -0.505;
   1:L PR[91] R[100]mm/sec CNT100;
   1:  PR[GP1:91,1] = PR[GP1:90,1] + 33.346;
   1:  PR[GP1:91,2] = PR[GP1:90,2] + -0.338;
   1:L PR[91] R[100]mm/sec CNT100;
   1:  PR[GP1:91,1] = PR[GP1:90,1] + 32.662;
   1:  PR[GP1:91,2] = PR[GP1:90,2] + 4.687;
   1:L PR[91] R[100]mm/sec CNT100;
   1:  PR[GP1:91,1] = PR[GP1:90,1] + 32.585;
   1:  PR[GP1:91,2] = PR[GP1:90,2] + 5.360;
   1:L PR[91] R[100]mm/sec CNT100;
   1:  PR[GP1:91,1] = PR[GP1:90,1] + 30.330;
   1:  PR[GP1:91,2] = PR[GP1:90,2] + 10.572;
   1:L PR[91] R[100]mm/sec CNT100;
   1:  PR[GP1:91,1] = PR[GP1:90,1] + 30.029;
   1:  PR[GP1:91,2] = PR[GP1:90,2] + 10.968;
   1:L PR[91] R[100]mm/sec CNT100;
   1:  PR[GP1:91,1] = PR[GP1:90,1] + 26.719;
   1:  PR[GP1:91,2] = PR[GP1:90,2] + 15.157;
   1:L PR[91] R[100]mm/sec CNT100;
   1:  PR[GP1:91,1] = PR[GP1:90,1] + 26.102;
   1:  PR[GP1:91,2] = PR[GP1:90,2] + 15.640;
   1:L PR[91] R[100]mm/sec CNT100;
   1:  PR[GP1:91,1] = PR[GP1:90,1] + 21.994;
   1:  PR[GP1:91,2] = PR[GP1:90,2] + 18.693;
   1:L PR[91] R[100]mm/sec CNT100;
   1:  PR[GP1:91,1] = PR[GP1:90,1] + 20.941;
   1:  PR[GP1:91,2] = PR[GP1:90,2] + 19.152;
   1:L PR[91] R[100]mm/sec CNT100;
   1:  PR[GP1:91,1] = PR[GP1:90,1] + 16.462;
   1:  PR[GP1:91,2] = PR[GP1:90,2] + 20.964;
   1:L PR[91] R[100]mm/sec CNT100;
   1:  PR[GP1:91,1] = PR[GP1:90,1] + 14.938;
   1:  PR[GP1:91,2] = PR[GP1:90,2] + 21.208;
   1:L PR[91] R[100]mm/sec CNT100;
   1:  PR[GP1:91,1] = PR[GP1:90,1] + 10.498;
   1:  PR[GP1:91,2] = PR[GP1:90,2] + 21.792;
   1:L PR[91] R[100]mm/sec CNT100;
   1:  PR[GP1:91,1] = PR[GP1:90,1] + 8.535;
   1:  PR[GP1:91,2] = PR[GP1:90,2] + 21.602;
   1:L PR[91] R[100]mm/sec CNT100;
   1:  PR[GP1:91,1] = PR[GP1:90,1] + 4.473;
   1:  PR[GP1:91,2] = PR[GP1:90,2] + 21.090;
   1:L PR[91] R[100]mm/sec CNT100;
   1:  PR[GP1:91,1] = PR[GP1:90,1] + 3.875;
   1:  PR[GP1:91,2] = PR[GP1:90,2] + 20.895;
   1:L PR[91] R[100]mm/sec CNT100;
   1:  PR[GP1:91,1] = PR[GP1:90,1] + 1.263;
   1:  PR[GP1:91,2] = PR[GP1:90,2] + 19.937;
   1:L PR[91] R[100]mm/sec CNT100;
   1:  PR[GP1:91,1] = PR[GP1:90,1] + 0.599;
   1:  PR[GP1:91,2] = PR[GP1:90,2] + 19.630;
   1:L PR[91] R[100]mm/sec CNT100;
   1:  ! -- Layer/Ebene 78 -- !;
   1:  PR[91] = PR[90];
   1:  PR[GP1:91,1] = PR[GP1:90,1] + -0.531;
   1:  PR[GP1:91,2] = PR[GP1:90,2] + 20.009;
   1:  PR[GP1:91,3] = PR[GP1:90,3] + 47.885;
   1:L PR[91] R[100]mm/sec CNT100;
   1:  PR[GP1:91,1] = PR[GP1:90,1] + -0.783;
   1:  PR[GP1:91,2] = PR[GP1:90,2] + 20.005;
   1:L PR[91] R[100]mm/sec CNT100;
   1:  PR[GP1:91,1] = PR[GP1:90,1] + -3.712;
   1:  PR[GP1:91,2] = PR[GP1:90,2] + 21.073;
   1:L PR[91] R[100]mm/sec CNT100;
   1:  PR[GP1:91,1] = PR[GP1:90,1] + -4.097;
   1:  PR[GP1:91,2] = PR[GP1:90,2] + 21.197;
   1:L PR[91] R[100]mm/sec CNT100;
   1:  PR[GP1:91,1] = PR[GP1:90,1] + -7.917;
   1:  PR[GP1:91,2] = PR[GP1:90,2] + 21.676;
   1:L PR[91] R[100]mm/sec CNT100;
   1:  PR[GP1:91,1] = PR[GP1:90,1] + -10.144;
   1:  PR[GP1:91,2] = PR[GP1:90,2] + 21.891;
   1:L PR[91] R[100]mm/sec CNT100;
   1:  PR[GP1:91,1] = PR[GP1:90,1] + -14.334;
   1:  PR[GP1:91,2] = PR[GP1:90,2] + 21.341;
   1:L PR[91] R[100]mm/sec CNT100;
   1:  PR[GP1:91,1] = PR[GP1:90,1] + -16.122;
   1:  PR[GP1:91,2] = PR[GP1:90,2] + 21.054;
   1:L PR[91] R[100]mm/sec CNT100;
   1:  PR[GP1:91,1] = PR[GP1:90,1] + -20.362;
   1:  PR[GP1:91,2] = PR[GP1:90,2] + 19.338;
   1:L PR[91] R[100]mm/sec CNT100;
   1:  PR[GP1:91,1] = PR[GP1:90,1] + -21.667;
   1:  PR[GP1:91,2] = PR[GP1:90,2] + 18.768;
   1:L PR[91] R[100]mm/sec CNT100;
   1:  PR[GP1:91,1] = PR[GP1:90,1] + -25.564;
   1:  PR[GP1:91,2] = PR[GP1:90,2] + 15.871;
   1:L PR[91] R[100]mm/sec CNT100;
   1:  PR[GP1:91,1] = PR[GP1:90,1] + -26.401;
   1:  PR[GP1:91,2] = PR[GP1:90,2] + 15.216;
   1:L PR[91] R[100]mm/sec CNT100;
   1:  PR[GP1:91,1] = PR[GP1:90,1] + -29.548;
   1:  PR[GP1:91,2] = PR[GP1:90,2] + 11.240;
   1:L PR[91] R[100]mm/sec CNT100;
   1:  PR[GP1:91,1] = PR[GP1:90,1] + -30.019;
   1:  PR[GP1:91,2] = PR[GP1:90,2] + 10.621;
   1:L PR[91] R[100]mm/sec CNT100;
   1:  PR[GP1:91,1] = PR[GP1:90,1] + -32.060;
   1:  PR[GP1:91,2] = PR[GP1:90,2] + 5.899;
   1:L PR[91] R[100]mm/sec CNT100;
   1:  PR[GP1:91,1] = PR[GP1:90,1] + -32.282;
   1:  PR[GP1:91,2] = PR[GP1:90,2] + 5.363;
   1:L PR[91] R[100]mm/sec CNT100;
   1:  PR[GP1:91,1] = PR[GP1:90,1] + -32.987;
   1:  PR[GP1:91,2] = PR[GP1:90,2] + 0.161;
   1:L PR[91] R[100]mm/sec CNT100;
   1:  PR[GP1:91,1] = PR[GP1:90,1] + -33.031;
   1:  PR[GP1:91,2] = PR[GP1:90,2] + -0.285;
   1:L PR[91] R[100]mm/sec CNT100;
   1:  PR[GP1:91,1] = PR[GP1:90,1] + -32.409;
   1:  PR[GP1:91,2] = PR[GP1:90,2] + -4.843;
   1:L PR[91] R[100]mm/sec CNT100;
   1:  PR[GP1:91,1] = PR[GP1:90,1] + -32.350;
   1:  PR[GP1:91,2] = PR[GP1:90,2] + -5.456;
   1:L PR[91] R[100]mm/sec CNT100;
   1:  PR[GP1:91,1] = PR[GP1:90,1] + -32.279;
   1:  PR[GP1:91,2] = PR[GP1:90,2] + -5.996;
   1:L PR[91] R[100]mm/sec CNT100;
   1:  PR[GP1:91,1] = PR[GP1:90,1] + -32.058;
   1:  PR[GP1:91,2] = PR[GP1:90,2] + -6.530;
   1:L PR[91] R[100]mm/sec CNT100;
   1:  PR[GP1:91,1] = PR[GP1:90,1] + -30.011;
   1:  PR[GP1:91,2] = PR[GP1:90,2] + -11.257;
   1:L PR[91] R[100]mm/sec CNT100;
   1:  PR[GP1:91,1] = PR[GP1:90,1] + -29.540;
   1:  PR[GP1:91,2] = PR[GP1:90,2] + -11.877;
   1:L PR[91] R[100]mm/sec CNT100;
   1:  PR[GP1:91,1] = PR[GP1:90,1] + -26.386;
   1:  PR[GP1:91,2] = PR[GP1:90,2] + -15.855;
   1:L PR[91] R[100]mm/sec CNT100;
   1:  PR[GP1:91,1] = PR[GP1:90,1] + -25.547;
   1:  PR[GP1:91,2] = PR[GP1:90,2] + -16.511;
   1:L PR[91] R[100]mm/sec CNT100;
   1:  PR[GP1:91,1] = PR[GP1:90,1] + -21.642;
   1:  PR[GP1:91,2] = PR[GP1:90,2] + -19.406;
   1:L PR[91] R[100]mm/sec CNT100;
   1:  PR[GP1:91,1] = PR[GP1:90,1] + -20.333;
   1:  PR[GP1:91,2] = PR[GP1:90,2] + -19.976;
   1:L PR[91] R[100]mm/sec CNT100;
   1:  PR[GP1:91,1] = PR[GP1:90,1] + -16.088;
   1:  PR[GP1:91,2] = PR[GP1:90,2] + -21.688;
   1:L PR[91] R[100]mm/sec CNT100;
   1:  PR[GP1:91,1] = PR[GP1:90,1] + -14.296;
   1:  PR[GP1:91,2] = PR[GP1:90,2] + -21.972;
   1:L PR[91] R[100]mm/sec CNT100;
   1:  PR[GP1:91,1] = PR[GP1:90,1] + -10.103;
   1:  PR[GP1:91,2] = PR[GP1:90,2] + -22.515;
   1:L PR[91] R[100]mm/sec CNT100;
   1:  PR[GP1:91,1] = PR[GP1:90,1] + -7.851;
   1:  PR[GP1:91,2] = PR[GP1:90,2] + -22.293;
   1:L PR[91] R[100]mm/sec CNT100;
   1:  PR[GP1:91,1] = PR[GP1:90,1] + -4.067;
   1:  PR[GP1:91,2] = PR[GP1:90,2] + -21.809;
   1:L PR[91] R[100]mm/sec CNT100;
   1:  PR[GP1:91,1] = PR[GP1:90,1] + -1.865;
   1:  PR[GP1:91,2] = PR[GP1:90,2] + -21.042;
   1:L PR[91] R[100]mm/sec CNT100;
   1:  PR[GP1:91,1] = PR[GP1:90,1] + -0.903;
   1:  PR[GP1:91,2] = PR[GP1:90,2] + -20.665;
   1:L PR[91] R[100]mm/sec CNT100;
   1:  PR[GP1:91,1] = PR[GP1:90,1] + 0.680;
   1:  PR[GP1:91,2] = PR[GP1:90,2] + -20.453;
   1:L PR[91] R[100]mm/sec CNT100;
   1:  PR[GP1:91,1] = PR[GP1:90,1] + 1.182;
   1:  PR[GP1:91,2] = PR[GP1:90,2] + -20.722;
   1:L PR[91] R[100]mm/sec CNT100;
   1:  PR[GP1:91,1] = PR[GP1:90,1] + 2.022;
   1:  PR[GP1:91,2] = PR[GP1:90,2] + -21.042;
   1:L PR[91] R[100]mm/sec CNT100;
   1:  PR[GP1:91,1] = PR[GP1:90,1] + 3.549;
   1:  PR[GP1:91,2] = PR[GP1:90,2] + -21.590;
   1:L PR[91] R[100]mm/sec CNT100;
   1:  PR[GP1:91,1] = PR[GP1:90,1] + 3.964;
   1:  PR[GP1:91,2] = PR[GP1:90,2] + -21.728;
   1:L PR[91] R[100]mm/sec CNT100;
   1:  PR[GP1:91,1] = PR[GP1:90,1] + 7.580;
   1:  PR[GP1:91,2] = PR[GP1:90,2] + -22.196;
   1:L PR[91] R[100]mm/sec CNT100;
   1:  PR[GP1:91,1] = PR[GP1:90,1] + 8.065;
   1:  PR[GP1:91,2] = PR[GP1:90,2] + -22.299;
   1:L PR[91] R[100]mm/sec CNT100;
   1:  PR[GP1:91,1] = PR[GP1:90,1] + 10.258;
   1:  PR[GP1:91,2] = PR[GP1:90,2] + -22.516;
   1:L PR[91] R[100]mm/sec CNT100;
   1:  PR[GP1:91,1] = PR[GP1:90,1] + 14.451;
   1:  PR[GP1:91,2] = PR[GP1:90,2] + -21.972;
   1:L PR[91] R[100]mm/sec CNT100;
   1:  PR[GP1:91,1] = PR[GP1:90,1] + 16.244;
   1:  PR[GP1:91,2] = PR[GP1:90,2] + -21.687;
   1:L PR[91] R[100]mm/sec CNT100;
   1:  PR[GP1:91,1] = PR[GP1:90,1] + 20.490;
   1:  PR[GP1:91,2] = PR[GP1:90,2] + -19.977;
   1:L PR[91] R[100]mm/sec CNT100;
   1:  PR[GP1:91,1] = PR[GP1:90,1] + 21.798;
   1:  PR[GP1:91,2] = PR[GP1:90,2] + -19.408;
   1:L PR[91] R[100]mm/sec CNT100;
   1:  PR[GP1:91,1] = PR[GP1:90,1] + 25.703;
   1:  PR[GP1:91,2] = PR[GP1:90,2] + -16.512;
   1:L PR[91] R[100]mm/sec CNT100;
   1:  PR[GP1:91,1] = PR[GP1:90,1] + 26.541;
   1:  PR[GP1:91,2] = PR[GP1:90,2] + -15.857;
   1:L PR[91] R[100]mm/sec CNT100;
   1:  PR[GP1:91,1] = PR[GP1:90,1] + 29.696;
   1:  PR[GP1:91,2] = PR[GP1:90,2] + -11.872;
   1:L PR[91] R[100]mm/sec CNT100;
   1:  PR[GP1:91,1] = PR[GP1:90,1] + 30.168;
   1:  PR[GP1:91,2] = PR[GP1:90,2] + -11.250;
   1:L PR[91] R[100]mm/sec CNT100;
   1:  PR[GP1:91,1] = PR[GP1:90,1] + 32.215;
   1:  PR[GP1:91,2] = PR[GP1:90,2] + -6.543;
   1:L PR[91] R[100]mm/sec CNT100;
   1:  PR[GP1:91,1] = PR[GP1:90,1] + 32.436;
   1:  PR[GP1:91,2] = PR[GP1:90,2] + -6.009;
   1:L PR[91] R[100]mm/sec CNT100;
   1:  PR[GP1:91,1] = PR[GP1:90,1] + 33.143;
   1:  PR[GP1:91,2] = PR[GP1:90,2] + -0.786;
   1:L PR[91] R[100]mm/sec CNT100;
   1:  PR[GP1:91,1] = PR[GP1:90,1] + 33.188;
   1:  PR[GP1:91,2] = PR[GP1:90,2] + -0.338;
   1:L PR[91] R[100]mm/sec CNT100;
   1:  PR[GP1:91,1] = PR[GP1:90,1] + 32.567;
   1:  PR[GP1:91,2] = PR[GP1:90,2] + 4.228;
   1:L PR[91] R[100]mm/sec CNT100;
   1:  PR[GP1:91,1] = PR[GP1:90,1] + 32.508;
   1:  PR[GP1:91,2] = PR[GP1:90,2] + 4.841;
   1:L PR[91] R[100]mm/sec CNT100;
   1:  PR[GP1:91,1] = PR[GP1:90,1] + 32.437;
   1:  PR[GP1:91,2] = PR[GP1:90,2] + 5.381;
   1:L PR[91] R[100]mm/sec CNT100;
   1:  PR[GP1:91,1] = PR[GP1:90,1] + 32.217;
   1:  PR[GP1:91,2] = PR[GP1:90,2] + 5.912;
   1:L PR[91] R[100]mm/sec CNT100;
   1:  PR[GP1:91,1] = PR[GP1:90,1] + 30.175;
   1:  PR[GP1:91,2] = PR[GP1:90,2] + 10.614;
   1:L PR[91] R[100]mm/sec CNT100;
   1:  PR[GP1:91,1] = PR[GP1:90,1] + 29.704;
   1:  PR[GP1:91,2] = PR[GP1:90,2] + 11.235;
   1:L PR[91] R[100]mm/sec CNT100;
   1:  PR[GP1:91,1] = PR[GP1:90,1] + 26.556;
   1:  PR[GP1:91,2] = PR[GP1:90,2] + 15.218;
   1:L PR[91] R[100]mm/sec CNT100;
   1:  PR[GP1:91,1] = PR[GP1:90,1] + 25.720;
   1:  PR[GP1:91,2] = PR[GP1:90,2] + 15.873;
   1:L PR[91] R[100]mm/sec CNT100;
   1:  PR[GP1:91,1] = PR[GP1:90,1] + 21.822;
   1:  PR[GP1:91,2] = PR[GP1:90,2] + 18.770;
   1:L PR[91] R[100]mm/sec CNT100;
   1:  PR[GP1:91,1] = PR[GP1:90,1] + 20.517;
   1:  PR[GP1:91,2] = PR[GP1:90,2] + 19.339;
   1:L PR[91] R[100]mm/sec CNT100;
   1:  PR[GP1:91,1] = PR[GP1:90,1] + 16.277;
   1:  PR[GP1:91,2] = PR[GP1:90,2] + 21.054;
   1:L PR[91] R[100]mm/sec CNT100;
   1:  PR[GP1:91,1] = PR[GP1:90,1] + 14.489;
   1:  PR[GP1:91,2] = PR[GP1:90,2] + 21.341;
   1:L PR[91] R[100]mm/sec CNT100;
   1:  PR[GP1:91,1] = PR[GP1:90,1] + 10.299;
   1:  PR[GP1:91,2] = PR[GP1:90,2] + 21.891;
   1:L PR[91] R[100]mm/sec CNT100;
   1:  PR[GP1:91,1] = PR[GP1:90,1] + 8.073;
   1:  PR[GP1:91,2] = PR[GP1:90,2] + 21.677;
   1:L PR[91] R[100]mm/sec CNT100;
   1:  PR[GP1:91,1] = PR[GP1:90,1] + 4.257;
   1:  PR[GP1:91,2] = PR[GP1:90,2] + 21.195;
   1:L PR[91] R[100]mm/sec CNT100;
   1:  PR[GP1:91,1] = PR[GP1:90,1] + 3.582;
   1:  PR[GP1:91,2] = PR[GP1:90,2] + 20.975;
   1:L PR[91] R[100]mm/sec CNT100;
   1:  PR[GP1:91,1] = PR[GP1:90,1] + 1.247;
   1:  PR[GP1:91,2] = PR[GP1:90,2] + 20.119;
   1:L PR[91] R[100]mm/sec CNT100;
   1:  PR[GP1:91,1] = PR[GP1:90,1] + 0.615;
   1:  PR[GP1:91,2] = PR[GP1:90,2] + 19.826;
   1:L PR[91] R[100]mm/sec CNT100;
   1:  ! -- Layer/Ebene 79 -- !;
   1:  PR[91] = PR[90];
   1:  PR[GP1:91,1] = PR[GP1:90,1] + -0.417;
   1:  PR[GP1:91,2] = PR[GP1:90,2] + 20.191;
   1:  PR[GP1:91,3] = PR[GP1:90,3] + 48.495;
   1:L PR[91] R[100]mm/sec CNT100;
   1:  PR[GP1:91,1] = PR[GP1:90,1] + -0.767;
   1:  PR[GP1:91,2] = PR[GP1:90,2] + 20.186;
   1:L PR[91] R[100]mm/sec CNT100;
   1:  PR[GP1:91,1] = PR[GP1:90,1] + -3.445;
   1:  PR[GP1:91,2] = PR[GP1:90,2] + 21.162;
   1:L PR[91] R[100]mm/sec CNT100;
   1:  PR[GP1:91,1] = PR[GP1:90,1] + -3.881;
   1:  PR[GP1:91,2] = PR[GP1:90,2] + 21.302;
   1:L PR[91] R[100]mm/sec CNT100;
   1:  PR[GP1:91,1] = PR[GP1:90,1] + -7.455;
   1:  PR[GP1:91,2] = PR[GP1:90,2] + 21.750;
   1:L PR[91] R[100]mm/sec CNT100;
   1:  PR[GP1:91,1] = PR[GP1:90,1] + -9.945;
   1:  PR[GP1:91,2] = PR[GP1:90,2] + 21.991;
   1:L PR[91] R[100]mm/sec CNT100;
   1:  PR[GP1:91,1] = PR[GP1:90,1] + -13.885;
   1:  PR[GP1:91,2] = PR[GP1:90,2] + 21.473;
   1:L PR[91] R[100]mm/sec CNT100;
   1:  PR[GP1:91,1] = PR[GP1:90,1] + -15.938;
   1:  PR[GP1:91,2] = PR[GP1:90,2] + 21.144;
   1:L PR[91] R[100]mm/sec CNT100;
   1:  PR[GP1:91,1] = PR[GP1:90,1] + -19.937;
   1:  PR[GP1:91,2] = PR[GP1:90,2] + 19.525;
   1:L PR[91] R[100]mm/sec CNT100;
   1:  PR[GP1:91,1] = PR[GP1:90,1] + -21.495;
   1:  PR[GP1:91,2] = PR[GP1:90,2] + 18.845;
   1:L PR[91] R[100]mm/sec CNT100;
   1:  PR[GP1:91,1] = PR[GP1:90,1] + -25.182;
   1:  PR[GP1:91,2] = PR[GP1:90,2] + 16.105;
   1:L PR[91] R[100]mm/sec CNT100;
   1:  PR[GP1:91,1] = PR[GP1:90,1] + -26.239;
   1:  PR[GP1:91,2] = PR[GP1:90,2] + 15.277;
   1:L PR[91] R[100]mm/sec CNT100;
   1:  PR[GP1:91,1] = PR[GP1:90,1] + -29.222;
   1:  PR[GP1:91,2] = PR[GP1:90,2] + 11.508;
   1:L PR[91] R[100]mm/sec CNT100;
   1:  PR[GP1:91,1] = PR[GP1:90,1] + -29.864;
   1:  PR[GP1:91,2] = PR[GP1:90,2] + 10.663;
   1:L PR[91] R[100]mm/sec CNT100;
   1:  PR[GP1:91,1] = PR[GP1:90,1] + -31.802;
   1:  PR[GP1:91,2] = PR[GP1:90,2] + 6.180;
   1:L PR[91] R[100]mm/sec CNT100;
   1:  PR[GP1:91,1] = PR[GP1:90,1] + -32.131;
   1:  PR[GP1:91,2] = PR[GP1:90,2] + 5.384;
   1:L PR[91] R[100]mm/sec CNT100;
   1:  PR[GP1:91,1] = PR[GP1:90,1] + -32.801;
   1:  PR[GP1:91,2] = PR[GP1:90,2] + 0.442;
   1:L PR[91] R[100]mm/sec CNT100;
   1:  PR[GP1:91,1] = PR[GP1:90,1] + -32.873;
   1:  PR[GP1:91,2] = PR[GP1:90,2] + -0.285;
   1:L PR[91] R[100]mm/sec CNT100;
   1:  PR[GP1:91,1] = PR[GP1:90,1] + -32.315;
   1:  PR[GP1:91,2] = PR[GP1:90,2] + -4.371;
   1:L PR[91] R[100]mm/sec CNT100;
   1:  PR[GP1:91,1] = PR[GP1:90,1] + -32.236;
   1:  PR[GP1:91,2] = PR[GP1:90,2] + -5.204;
   1:L PR[91] R[100]mm/sec CNT100;
   1:  PR[GP1:91,1] = PR[GP1:90,1] + -32.128;
   1:  PR[GP1:91,2] = PR[GP1:90,2] + -6.018;
   1:L PR[91] R[100]mm/sec CNT100;
   1:  PR[GP1:91,1] = PR[GP1:90,1] + -31.799;
   1:  PR[GP1:91,2] = PR[GP1:90,2] + -6.812;
   1:L PR[91] R[100]mm/sec CNT100;
   1:  PR[GP1:91,1] = PR[GP1:90,1] + -29.856;
   1:  PR[GP1:91,2] = PR[GP1:90,2] + -11.299;
   1:L PR[91] R[100]mm/sec CNT100;
   1:  PR[GP1:91,1] = PR[GP1:90,1] + -29.213;
   1:  PR[GP1:91,2] = PR[GP1:90,2] + -12.145;
   1:L PR[91] R[100]mm/sec CNT100;
   1:  PR[GP1:91,1] = PR[GP1:90,1] + -26.224;
   1:  PR[GP1:91,2] = PR[GP1:90,2] + -15.915;
   1:L PR[91] R[100]mm/sec CNT100;
   1:  PR[GP1:91,1] = PR[GP1:90,1] + -25.164;
   1:  PR[GP1:91,2] = PR[GP1:90,2] + -16.744;
   1:L PR[91] R[100]mm/sec CNT100;
   1:  PR[GP1:91,1] = PR[GP1:90,1] + -21.470;
   1:  PR[GP1:91,2] = PR[GP1:90,2] + -19.483;
   1:L PR[91] R[100]mm/sec CNT100;
   1:  PR[GP1:91,1] = PR[GP1:90,1] + -19.909;
   1:  PR[GP1:91,2] = PR[GP1:90,2] + -20.163;
   1:L PR[91] R[100]mm/sec CNT100;
   1:  PR[GP1:91,1] = PR[GP1:90,1] + -15.904;
   1:  PR[GP1:91,2] = PR[GP1:90,2] + -21.778;
   1:L PR[91] R[100]mm/sec CNT100;
   1:  PR[GP1:91,1] = PR[GP1:90,1] + -13.847;
   1:  PR[GP1:91,2] = PR[GP1:90,2] + -22.104;
   1:L PR[91] R[100]mm/sec CNT100;
   1:  PR[GP1:91,1] = PR[GP1:90,1] + -9.904;
   1:  PR[GP1:91,2] = PR[GP1:90,2] + -22.615;
   1:L PR[91] R[100]mm/sec CNT100;
   1:  PR[GP1:91,1] = PR[GP1:90,1] + -7.386;
   1:  PR[GP1:91,2] = PR[GP1:90,2] + -22.366;
   1:L PR[91] R[100]mm/sec CNT100;
   1:  PR[GP1:91,1] = PR[GP1:90,1] + -3.850;
   1:  PR[GP1:91,2] = PR[GP1:90,2] + -21.914;
   1:L PR[91] R[100]mm/sec CNT100;
   1:  PR[GP1:91,1] = PR[GP1:90,1] + -1.430;
   1:  PR[GP1:91,2] = PR[GP1:90,2] + -21.071;
   1:L PR[91] R[100]mm/sec CNT100;
   1:  PR[GP1:91,1] = PR[GP1:90,1] + -0.883;
   1:  PR[GP1:91,2] = PR[GP1:90,2] + -20.857;
   1:L PR[91] R[100]mm/sec CNT100;
   1:  PR[GP1:91,1] = PR[GP1:90,1] + 0.701;
   1:  PR[GP1:91,2] = PR[GP1:90,2] + -20.652;
   1:L PR[91] R[100]mm/sec CNT100;
   1:  PR[GP1:91,1] = PR[GP1:90,1] + 1.223;
   1:  PR[GP1:91,2] = PR[GP1:90,2] + -20.932;
   1:L PR[91] R[100]mm/sec CNT100;
   1:  PR[GP1:91,1] = PR[GP1:90,1] + 1.587;
   1:  PR[GP1:91,2] = PR[GP1:90,2] + -21.071;
   1:L PR[91] R[100]mm/sec CNT100;
   1:  PR[GP1:91,1] = PR[GP1:90,1] + 3.258;
   1:  PR[GP1:91,2] = PR[GP1:90,2] + -21.671;
   1:L PR[91] R[100]mm/sec CNT100;
   1:  PR[GP1:91,1] = PR[GP1:90,1] + 3.725;
   1:  PR[GP1:91,2] = PR[GP1:90,2] + -21.826;
   1:L PR[91] R[100]mm/sec CNT100;
   1:  PR[GP1:91,1] = PR[GP1:90,1] + 7.061;
   1:  PR[GP1:91,2] = PR[GP1:90,2] + -22.258;
   1:L PR[91] R[100]mm/sec CNT100;
   1:  PR[GP1:91,1] = PR[GP1:90,1] + 7.601;
   1:  PR[GP1:91,2] = PR[GP1:90,2] + -22.372;
   1:L PR[91] R[100]mm/sec CNT100;
   1:  PR[GP1:91,1] = PR[GP1:90,1] + 10.059;
   1:  PR[GP1:91,2] = PR[GP1:90,2] + -22.615;
   1:L PR[91] R[100]mm/sec CNT100;
   1:  PR[GP1:91,1] = PR[GP1:90,1] + 14.002;
   1:  PR[GP1:91,2] = PR[GP1:90,2] + -22.104;
   1:L PR[91] R[100]mm/sec CNT100;
   1:  PR[GP1:91,1] = PR[GP1:90,1] + 16.060;
   1:  PR[GP1:91,2] = PR[GP1:90,2] + -21.777;
   1:L PR[91] R[100]mm/sec CNT100;
   1:  PR[GP1:91,1] = PR[GP1:90,1] + 20.065;
   1:  PR[GP1:91,2] = PR[GP1:90,2] + -20.163;
   1:L PR[91] R[100]mm/sec CNT100;
   1:  PR[GP1:91,1] = PR[GP1:90,1] + 21.626;
   1:  PR[GP1:91,2] = PR[GP1:90,2] + -19.485;
   1:L PR[91] R[100]mm/sec CNT100;
   1:  PR[GP1:91,1] = PR[GP1:90,1] + 25.320;
   1:  PR[GP1:91,2] = PR[GP1:90,2] + -16.746;
   1:L PR[91] R[100]mm/sec CNT100;
   1:  PR[GP1:91,1] = PR[GP1:90,1] + 26.379;
   1:  PR[GP1:91,2] = PR[GP1:90,2] + -15.917;
   1:L PR[91] R[100]mm/sec CNT100;
   1:  PR[GP1:91,1] = PR[GP1:90,1] + 29.369;
   1:  PR[GP1:91,2] = PR[GP1:90,2] + -12.140;
   1:L PR[91] R[100]mm/sec CNT100;
   1:  PR[GP1:91,1] = PR[GP1:90,1] + 30.013;
   1:  PR[GP1:91,2] = PR[GP1:90,2] + -11.293;
   1:L PR[91] R[100]mm/sec CNT100;
   1:  PR[GP1:91,1] = PR[GP1:90,1] + 31.956;
   1:  PR[GP1:91,2] = PR[GP1:90,2] + -6.824;
   1:L PR[91] R[100]mm/sec CNT100;
   1:  PR[GP1:91,1] = PR[GP1:90,1] + 32.286;
   1:  PR[GP1:91,2] = PR[GP1:90,2] + -6.030;
   1:L PR[91] R[100]mm/sec CNT100;
   1:  PR[GP1:91,1] = PR[GP1:90,1] + 32.958;
   1:  PR[GP1:91,2] = PR[GP1:90,2] + -1.067;
   1:L PR[91] R[100]mm/sec CNT100;
   1:  PR[GP1:91,1] = PR[GP1:90,1] + 33.030;
   1:  PR[GP1:91,2] = PR[GP1:90,2] + -0.338;
   1:L PR[91] R[100]mm/sec CNT100;
   1:  PR[GP1:91,1] = PR[GP1:90,1] + 32.473;
   1:  PR[GP1:91,2] = PR[GP1:90,2] + 3.755;
   1:L PR[91] R[100]mm/sec CNT100;
   1:  PR[GP1:91,1] = PR[GP1:90,1] + 32.394;
   1:  PR[GP1:91,2] = PR[GP1:90,2] + 4.589;
   1:L PR[91] R[100]mm/sec CNT100;
   1:  PR[GP1:91,1] = PR[GP1:90,1] + 32.287;
   1:  PR[GP1:91,2] = PR[GP1:90,2] + 5.402;
   1:L PR[91] R[100]mm/sec CNT100;
   1:  PR[GP1:91,1] = PR[GP1:90,1] + 31.959;
   1:  PR[GP1:91,2] = PR[GP1:90,2] + 6.193;
   1:L PR[91] R[100]mm/sec CNT100;
   1:  PR[GP1:91,1] = PR[GP1:90,1] + 30.020;
   1:  PR[GP1:91,2] = PR[GP1:90,2] + 10.657;
   1:L PR[91] R[100]mm/sec CNT100;
   1:  PR[GP1:91,1] = PR[GP1:90,1] + 29.378;
   1:  PR[GP1:91,2] = PR[GP1:90,2] + 11.503;
   1:L PR[91] R[100]mm/sec CNT100;
   1:  PR[GP1:91,1] = PR[GP1:90,1] + 26.394;
   1:  PR[GP1:91,2] = PR[GP1:90,2] + 15.279;
   1:L PR[91] R[100]mm/sec CNT100;
   1:  PR[GP1:91,1] = PR[GP1:90,1] + 25.338;
   1:  PR[GP1:91,2] = PR[GP1:90,2] + 16.106;
   1:L PR[91] R[100]mm/sec CNT100;
   1:  PR[GP1:91,1] = PR[GP1:90,1] + 21.650;
   1:  PR[GP1:91,2] = PR[GP1:90,2] + 18.847;
   1:L PR[91] R[100]mm/sec CNT100;
   1:  PR[GP1:91,1] = PR[GP1:90,1] + 20.093;
   1:  PR[GP1:91,2] = PR[GP1:90,2] + 19.526;
   1:L PR[91] R[100]mm/sec CNT100;
   1:  PR[GP1:91,1] = PR[GP1:90,1] + 16.093;
   1:  PR[GP1:91,2] = PR[GP1:90,2] + 21.144;
   1:L PR[91] R[100]mm/sec CNT100;
   1:  PR[GP1:91,1] = PR[GP1:90,1] + 14.040;
   1:  PR[GP1:91,2] = PR[GP1:90,2] + 21.473;
   1:L PR[91] R[100]mm/sec CNT100;
   1:  PR[GP1:91,1] = PR[GP1:90,1] + 10.100;
   1:  PR[GP1:91,2] = PR[GP1:90,2] + 21.991;
   1:L PR[91] R[100]mm/sec CNT100;
   1:  PR[GP1:91,1] = PR[GP1:90,1] + 7.610;
   1:  PR[GP1:91,2] = PR[GP1:90,2] + 21.751;
   1:L PR[91] R[100]mm/sec CNT100;
   1:  PR[GP1:91,1] = PR[GP1:90,1] + 4.040;
   1:  PR[GP1:91,2] = PR[GP1:90,2] + 21.301;
   1:L PR[91] R[100]mm/sec CNT100;
   1:  PR[GP1:91,1] = PR[GP1:90,1] + 3.289;
   1:  PR[GP1:91,2] = PR[GP1:90,2] + 21.056;
   1:L PR[91] R[100]mm/sec CNT100;
   1:  PR[GP1:91,1] = PR[GP1:90,1] + 1.232;
   1:  PR[GP1:91,2] = PR[GP1:90,2] + 20.301;
   1:L PR[91] R[100]mm/sec CNT100;
   1:  PR[GP1:91,1] = PR[GP1:90,1] + 0.632;
   1:  PR[GP1:91,2] = PR[GP1:90,2] + 20.024;
   1:L PR[91] R[100]mm/sec CNT100;
   1:  ! -- Layer/Ebene 80 -- !;
   1:  PR[91] = PR[90];
   1:  PR[GP1:91,1] = PR[GP1:90,1] + -0.304;
   1:  PR[GP1:91,2] = PR[GP1:90,2] + 20.373;
   1:  PR[GP1:91,3] = PR[GP1:90,3] + 49.105;
   1:L PR[91] R[100]mm/sec CNT100;
   1:  PR[GP1:91,1] = PR[GP1:90,1] + -0.751;
   1:  PR[GP1:91,2] = PR[GP1:90,2] + 20.366;
   1:L PR[91] R[100]mm/sec CNT100;
   1:  PR[GP1:91,1] = PR[GP1:90,1] + -3.178;
   1:  PR[GP1:91,2] = PR[GP1:90,2] + 21.251;
   1:L PR[91] R[100]mm/sec CNT100;
   1:  PR[GP1:91,1] = PR[GP1:90,1] + -3.664;
   1:  PR[GP1:91,2] = PR[GP1:90,2] + 21.407;
   1:L PR[91] R[100]mm/sec CNT100;
   1:  PR[GP1:91,1] = PR[GP1:90,1] + -6.992;
   1:  PR[GP1:91,2] = PR[GP1:90,2] + 21.825;
   1:L PR[91] R[100]mm/sec CNT100;
   1:  PR[GP1:91,1] = PR[GP1:90,1] + -9.746;
   1:  PR[GP1:91,2] = PR[GP1:90,2] + 22.090;
   1:L PR[91] R[100]mm/sec CNT100;
   1:  PR[GP1:91,1] = PR[GP1:90,1] + -13.436;
   1:  PR[GP1:91,2] = PR[GP1:90,2] + 21.606;
   1:L PR[91] R[100]mm/sec CNT100;
   1:  PR[GP1:91,1] = PR[GP1:90,1] + -15.753;
   1:  PR[GP1:91,2] = PR[GP1:90,2] + 21.234;
   1:L PR[91] R[100]mm/sec CNT100;
   1:  PR[GP1:91,1] = PR[GP1:90,1] + -19.513;
   1:  PR[GP1:91,2] = PR[GP1:90,2] + 19.712;
   1:L PR[91] R[100]mm/sec CNT100;
   1:  PR[GP1:91,1] = PR[GP1:90,1] + -21.322;
   1:  PR[GP1:91,2] = PR[GP1:90,2] + 18.922;
   1:L PR[91] R[100]mm/sec CNT100;
   1:  PR[GP1:91,1] = PR[GP1:90,1] + -24.799;
   1:  PR[GP1:91,2] = PR[GP1:90,2] + 16.338;
   1:L PR[91] R[100]mm/sec CNT100;
   1:  PR[GP1:91,1] = PR[GP1:90,1] + -26.077;
   1:  PR[GP1:91,2] = PR[GP1:90,2] + 15.337;
   1:L PR[91] R[100]mm/sec CNT100;
   1:  PR[GP1:91,1] = PR[GP1:90,1] + -28.896;
   1:  PR[GP1:91,2] = PR[GP1:90,2] + 11.775;
   1:L PR[91] R[100]mm/sec CNT100;
   1:  PR[GP1:91,1] = PR[GP1:90,1] + -29.709;
   1:  PR[GP1:91,2] = PR[GP1:90,2] + 10.706;
   1:L PR[91] R[100]mm/sec CNT100;
   1:  PR[GP1:91,1] = PR[GP1:90,1] + -31.544;
   1:  PR[GP1:91,2] = PR[GP1:90,2] + 6.462;
   1:L PR[91] R[100]mm/sec CNT100;
   1:  PR[GP1:91,1] = PR[GP1:90,1] + -31.981;
   1:  PR[GP1:91,2] = PR[GP1:90,2] + 5.405;
   1:L PR[91] R[100]mm/sec CNT100;
   1:  PR[GP1:91,1] = PR[GP1:90,1] + -32.615;
   1:  PR[GP1:91,2] = PR[GP1:90,2] + 0.723;
   1:L PR[91] R[100]mm/sec CNT100;
   1:  PR[GP1:91,1] = PR[GP1:90,1] + -32.715;
   1:  PR[GP1:91,2] = PR[GP1:90,2] + -0.285;
   1:L PR[91] R[100]mm/sec CNT100;
   1:  PR[GP1:91,1] = PR[GP1:90,1] + -32.222;
   1:  PR[GP1:91,2] = PR[GP1:90,2] + -3.899;
   1:L PR[91] R[100]mm/sec CNT100;
   1:  PR[GP1:91,1] = PR[GP1:90,1] + -32.121;
   1:  PR[GP1:91,2] = PR[GP1:90,2] + -4.952;
   1:L PR[91] R[100]mm/sec CNT100;
   1:  PR[GP1:91,1] = PR[GP1:90,1] + -31.978;
   1:  PR[GP1:91,2] = PR[GP1:90,2] + -6.039;
   1:L PR[91] R[100]mm/sec CNT100;
   1:  PR[GP1:91,1] = PR[GP1:90,1] + -31.541;
   1:  PR[GP1:91,2] = PR[GP1:90,2] + -7.093;
   1:L PR[91] R[100]mm/sec CNT100;
   1:  PR[GP1:91,1] = PR[GP1:90,1] + -29.702;
   1:  PR[GP1:91,2] = PR[GP1:90,2] + -11.342;
   1:L PR[91] R[100]mm/sec CNT100;
   1:  PR[GP1:91,1] = PR[GP1:90,1] + -28.887;
   1:  PR[GP1:91,2] = PR[GP1:90,2] + -12.412;
   1:L PR[91] R[100]mm/sec CNT100;
   1:  PR[GP1:91,1] = PR[GP1:90,1] + -26.062;
   1:  PR[GP1:91,2] = PR[GP1:90,2] + -15.976;
   1:L PR[91] R[100]mm/sec CNT100;
   1:  PR[GP1:91,1] = PR[GP1:90,1] + -24.781;
   1:  PR[GP1:91,2] = PR[GP1:90,2] + -16.977;
   1:L PR[91] R[100]mm/sec CNT100;
   1:  PR[GP1:91,1] = PR[GP1:90,1] + -21.298;
   1:  PR[GP1:91,2] = PR[GP1:90,2] + -19.560;
   1:L PR[91] R[100]mm/sec CNT100;
   1:  PR[GP1:91,1] = PR[GP1:90,1] + -19.485;
   1:  PR[GP1:91,2] = PR[GP1:90,2] + -20.349;
   1:L PR[91] R[100]mm/sec CNT100;
   1:  PR[GP1:91,1] = PR[GP1:90,1] + -15.719;
   1:  PR[GP1:91,2] = PR[GP1:90,2] + -21.867;
   1:L PR[91] R[100]mm/sec CNT100;
   1:  PR[GP1:91,1] = PR[GP1:90,1] + -13.398;
   1:  PR[GP1:91,2] = PR[GP1:90,2] + -22.236;
   1:L PR[91] R[100]mm/sec CNT100;
   1:  PR[GP1:91,1] = PR[GP1:90,1] + -9.705;
   1:  PR[GP1:91,2] = PR[GP1:90,2] + -22.715;
   1:L PR[91] R[100]mm/sec CNT100;
   1:  PR[GP1:91,1] = PR[GP1:90,1] + -6.922;
   1:  PR[GP1:91,2] = PR[GP1:90,2] + -22.439;
   1:L PR[91] R[100]mm/sec CNT100;
   1:  PR[GP1:91,1] = PR[GP1:90,1] + -3.633;
   1:  PR[GP1:91,2] = PR[GP1:90,2] + -22.019;
   1:L PR[91] R[100]mm/sec CNT100;
   1:  PR[GP1:91,1] = PR[GP1:90,1] + -0.832;
   1:  PR[GP1:91,2] = PR[GP1:90,2] + -21.045;
   1:L PR[91] R[100]mm/sec CNT100;
   1:  PR[GP1:91,1] = PR[GP1:90,1] + 0.721;
   1:  PR[GP1:91,2] = PR[GP1:90,2] + -20.851;
   1:L PR[91] R[100]mm/sec CNT100;
   1:  PR[GP1:91,1] = PR[GP1:90,1] + 1.251;
   1:  PR[GP1:91,2] = PR[GP1:90,2] + -21.135;
   1:L PR[91] R[100]mm/sec CNT100;
   1:  PR[GP1:91,1] = PR[GP1:90,1] + 2.967;
   1:  PR[GP1:91,2] = PR[GP1:90,2] + -21.752;
   1:L PR[91] R[100]mm/sec CNT100;
   1:  PR[GP1:91,1] = PR[GP1:90,1] + 3.486;
   1:  PR[GP1:91,2] = PR[GP1:90,2] + -21.924;
   1:L PR[91] R[100]mm/sec CNT100;
   1:  PR[GP1:91,1] = PR[GP1:90,1] + 6.541;
   1:  PR[GP1:91,2] = PR[GP1:90,2] + -22.319;
   1:L PR[91] R[100]mm/sec CNT100;
   1:  PR[GP1:91,1] = PR[GP1:90,1] + 7.136;
   1:  PR[GP1:91,2] = PR[GP1:90,2] + -22.445;
   1:L PR[91] R[100]mm/sec CNT100;
   1:  PR[GP1:91,1] = PR[GP1:90,1] + 9.861;
   1:  PR[GP1:91,2] = PR[GP1:90,2] + -22.715;
   1:L PR[91] R[100]mm/sec CNT100;
   1:  PR[GP1:91,1] = PR[GP1:90,1] + 13.553;
   1:  PR[GP1:91,2] = PR[GP1:90,2] + -22.236;
   1:L PR[91] R[100]mm/sec CNT100;
   1:  PR[GP1:91,1] = PR[GP1:90,1] + 15.875;
   1:  PR[GP1:91,2] = PR[GP1:90,2] + -21.867;
   1:L PR[91] R[100]mm/sec CNT100;
   1:  PR[GP1:91,1] = PR[GP1:90,1] + 19.641;
   1:  PR[GP1:91,2] = PR[GP1:90,2] + -20.350;
   1:L PR[91] R[100]mm/sec CNT100;
   1:  PR[GP1:91,1] = PR[GP1:90,1] + 21.454;
   1:  PR[GP1:91,2] = PR[GP1:90,2] + -19.562;
   1:L PR[91] R[100]mm/sec CNT100;
   1:  PR[GP1:91,1] = PR[GP1:90,1] + 24.938;
   1:  PR[GP1:91,2] = PR[GP1:90,2] + -16.979;
   1:L PR[91] R[100]mm/sec CNT100;
   1:  PR[GP1:91,1] = PR[GP1:90,1] + 26.217;
   1:  PR[GP1:91,2] = PR[GP1:90,2] + -15.978;
   1:L PR[91] R[100]mm/sec CNT100;
   1:  PR[GP1:91,1] = PR[GP1:90,1] + 29.043;
   1:  PR[GP1:91,2] = PR[GP1:90,2] + -12.407;
   1:L PR[91] R[100]mm/sec CNT100;
   1:  PR[GP1:91,1] = PR[GP1:90,1] + 29.858;
   1:  PR[GP1:91,2] = PR[GP1:90,2] + -11.335;
   1:L PR[91] R[100]mm/sec CNT100;
   1:  PR[GP1:91,1] = PR[GP1:90,1] + 31.698;
   1:  PR[GP1:91,2] = PR[GP1:90,2] + -7.104;
   1:L PR[91] R[100]mm/sec CNT100;
   1:  PR[GP1:91,1] = PR[GP1:90,1] + 32.136;
   1:  PR[GP1:91,2] = PR[GP1:90,2] + -6.050;
   1:L PR[91] R[100]mm/sec CNT100;
   1:  PR[GP1:91,1] = PR[GP1:90,1] + 32.772;
   1:  PR[GP1:91,2] = PR[GP1:90,2] + -1.349;
   1:L PR[91] R[100]mm/sec CNT100;
   1:  PR[GP1:91,1] = PR[GP1:90,1] + 32.872;
   1:  PR[GP1:91,2] = PR[GP1:90,2] + -0.338;
   1:L PR[91] R[100]mm/sec CNT100;
   1:  PR[GP1:91,1] = PR[GP1:90,1] + 32.380;
   1:  PR[GP1:91,2] = PR[GP1:90,2] + 3.282;
   1:L PR[91] R[100]mm/sec CNT100;
   1:  PR[GP1:91,1] = PR[GP1:90,1] + 32.279;
   1:  PR[GP1:91,2] = PR[GP1:90,2] + 4.337;
   1:L PR[91] R[100]mm/sec CNT100;
   1:  PR[GP1:91,1] = PR[GP1:90,1] + 32.136;
   1:  PR[GP1:91,2] = PR[GP1:90,2] + 5.422;
   1:L PR[91] R[100]mm/sec CNT100;
   1:  PR[GP1:91,1] = PR[GP1:90,1] + 31.701;
   1:  PR[GP1:91,2] = PR[GP1:90,2] + 6.473;
   1:L PR[91] R[100]mm/sec CNT100;
   1:  PR[GP1:91,1] = PR[GP1:90,1] + 29.865;
   1:  PR[GP1:91,2] = PR[GP1:90,2] + 10.699;
   1:L PR[91] R[100]mm/sec CNT100;
   1:  PR[GP1:91,1] = PR[GP1:90,1] + 29.052;
   1:  PR[GP1:91,2] = PR[GP1:90,2] + 11.770;
   1:L PR[91] R[100]mm/sec CNT100;
   1:  PR[GP1:91,1] = PR[GP1:90,1] + 26.232;
   1:  PR[GP1:91,2] = PR[GP1:90,2] + 15.339;
   1:L PR[91] R[100]mm/sec CNT100;
   1:  PR[GP1:91,1] = PR[GP1:90,1] + 24.955;
   1:  PR[GP1:91,2] = PR[GP1:90,2] + 16.340;
   1:L PR[91] R[100]mm/sec CNT100;
   1:  PR[GP1:91,1] = PR[GP1:90,1] + 21.478;
   1:  PR[GP1:91,2] = PR[GP1:90,2] + 18.924;
   1:L PR[91] R[100]mm/sec CNT100;
   1:  PR[GP1:91,1] = PR[GP1:90,1] + 19.669;
   1:  PR[GP1:91,2] = PR[GP1:90,2] + 19.713;
   1:L PR[91] R[100]mm/sec CNT100;
   1:  PR[GP1:91,1] = PR[GP1:90,1] + 15.908;
   1:  PR[GP1:91,2] = PR[GP1:90,2] + 21.234;
   1:L PR[91] R[100]mm/sec CNT100;
   1:  PR[GP1:91,1] = PR[GP1:90,1] + 13.591;
   1:  PR[GP1:91,2] = PR[GP1:90,2] + 21.606;
   1:L PR[91] R[100]mm/sec CNT100;
   1:  PR[GP1:91,1] = PR[GP1:90,1] + 9.901;
   1:  PR[GP1:91,2] = PR[GP1:90,2] + 22.090;
   1:L PR[91] R[100]mm/sec CNT100;
   1:  PR[GP1:91,1] = PR[GP1:90,1] + 7.148;
   1:  PR[GP1:91,2] = PR[GP1:90,2] + 21.825;
   1:L PR[91] R[100]mm/sec CNT100;
   1:  PR[GP1:91,1] = PR[GP1:90,1] + 3.824;
   1:  PR[GP1:91,2] = PR[GP1:90,2] + 21.406;
   1:L PR[91] R[100]mm/sec CNT100;
   1:  PR[GP1:91,1] = PR[GP1:90,1] + 2.996;
   1:  PR[GP1:91,2] = PR[GP1:90,2] + 21.136;
   1:L PR[91] R[100]mm/sec CNT100;
   1:  PR[GP1:91,1] = PR[GP1:90,1] + 1.216;
   1:  PR[GP1:91,2] = PR[GP1:90,2] + 20.483;
   1:L PR[91] R[100]mm/sec CNT100;
   1:  PR[GP1:91,1] = PR[GP1:90,1] + 0.649;
   1:  PR[GP1:91,2] = PR[GP1:90,2] + 20.221;
   1:L PR[91] R[100]mm/sec CNT100;
   1:  ! -- Layer/Ebene 81 -- !;
   1:  PR[91] = PR[90];
   1:  PR[GP1:91,1] = PR[GP1:90,1] + -0.191;
   1:  PR[GP1:91,2] = PR[GP1:90,2] + 20.555;
   1:  PR[GP1:91,3] = PR[GP1:90,3] + 49.715;
   1:L PR[91] R[100]mm/sec CNT100;
   1:  PR[GP1:91,1] = PR[GP1:90,1] + -0.735;
   1:  PR[GP1:91,2] = PR[GP1:90,2] + 20.547;
   1:L PR[91] R[100]mm/sec CNT100;
   1:  PR[GP1:91,1] = PR[GP1:90,1] + -2.912;
   1:  PR[GP1:91,2] = PR[GP1:90,2] + 21.340;
   1:L PR[91] R[100]mm/sec CNT100;
   1:  PR[GP1:91,1] = PR[GP1:90,1] + -3.447;
   1:  PR[GP1:91,2] = PR[GP1:90,2] + 21.512;
   1:L PR[91] R[100]mm/sec CNT100;
   1:  PR[GP1:91,1] = PR[GP1:90,1] + -6.529;
   1:  PR[GP1:91,2] = PR[GP1:90,2] + 21.899;
   1:L PR[91] R[100]mm/sec CNT100;
   1:  PR[GP1:91,1] = PR[GP1:90,1] + -9.546;
   1:  PR[GP1:91,2] = PR[GP1:90,2] + 22.190;
   1:L PR[91] R[100]mm/sec CNT100;
   1:  PR[GP1:91,1] = PR[GP1:90,1] + -12.986;
   1:  PR[GP1:91,2] = PR[GP1:90,2] + 21.738;
   1:L PR[91] R[100]mm/sec CNT100;
   1:  PR[GP1:91,1] = PR[GP1:90,1] + -15.568;
   1:  PR[GP1:91,2] = PR[GP1:90,2] + 21.324;
   1:L PR[91] R[100]mm/sec CNT100;
   1:  PR[GP1:91,1] = PR[GP1:90,1] + -19.088;
   1:  PR[GP1:91,2] = PR[GP1:90,2] + 19.899;
   1:L PR[91] R[100]mm/sec CNT100;
   1:  PR[GP1:91,1] = PR[GP1:90,1] + -21.150;
   1:  PR[GP1:91,2] = PR[GP1:90,2] + 18.999;
   1:L PR[91] R[100]mm/sec CNT100;
   1:  PR[GP1:91,1] = PR[GP1:90,1] + -24.417;
   1:  PR[GP1:91,2] = PR[GP1:90,2] + 16.571;
   1:L PR[91] R[100]mm/sec CNT100;
   1:  PR[GP1:91,1] = PR[GP1:90,1] + -25.914;
   1:  PR[GP1:91,2] = PR[GP1:90,2] + 15.398;
   1:L PR[91] R[100]mm/sec CNT100;
   1:  PR[GP1:91,1] = PR[GP1:90,1] + -28.571;
   1:  PR[GP1:91,2] = PR[GP1:90,2] + 12.042;
   1:L PR[91] R[100]mm/sec CNT100;
   1:  PR[GP1:91,1] = PR[GP1:90,1] + -29.554;
   1:  PR[GP1:91,2] = PR[GP1:90,2] + 10.748;
   1:L PR[91] R[100]mm/sec CNT100;
   1:  PR[GP1:91,1] = PR[GP1:90,1] + -31.285;
   1:  PR[GP1:91,2] = PR[GP1:90,2] + 6.743;
   1:L PR[91] R[100]mm/sec CNT100;
   1:  PR[GP1:91,1] = PR[GP1:90,1] + -31.830;
   1:  PR[GP1:91,2] = PR[GP1:90,2] + 5.427;
   1:L PR[91] R[100]mm/sec CNT100;
   1:  PR[GP1:91,1] = PR[GP1:90,1] + -32.430;
   1:  PR[GP1:91,2] = PR[GP1:90,2] + 1.004;
   1:L PR[91] R[100]mm/sec CNT100;
   1:  PR[GP1:91,1] = PR[GP1:90,1] + -32.557;
   1:  PR[GP1:91,2] = PR[GP1:90,2] + -0.285;
   1:L PR[91] R[100]mm/sec CNT100;
   1:  PR[GP1:91,1] = PR[GP1:90,1] + -32.129;
   1:  PR[GP1:91,2] = PR[GP1:90,2] + -3.427;
   1:L PR[91] R[100]mm/sec CNT100;
   1:  PR[GP1:91,1] = PR[GP1:90,1] + -32.007;
   1:  PR[GP1:91,2] = PR[GP1:90,2] + -4.700;
   1:L PR[91] R[100]mm/sec CNT100;
   1:  PR[GP1:91,1] = PR[GP1:90,1] + -31.827;
   1:  PR[GP1:91,2] = PR[GP1:90,2] + -6.060;
   1:L PR[91] R[100]mm/sec CNT100;
   1:  PR[GP1:91,1] = PR[GP1:90,1] + -31.282;
   1:  PR[GP1:91,2] = PR[GP1:90,2] + -7.375;
   1:L PR[91] R[100]mm/sec CNT100;
   1:  PR[GP1:91,1] = PR[GP1:90,1] + -29.547;
   1:  PR[GP1:91,2] = PR[GP1:90,2] + -11.384;
   1:L PR[91] R[100]mm/sec CNT100;
   1:  PR[GP1:91,1] = PR[GP1:90,1] + -28.561;
   1:  PR[GP1:91,2] = PR[GP1:90,2] + -12.680;
   1:L PR[91] R[100]mm/sec CNT100;
   1:  PR[GP1:91,1] = PR[GP1:90,1] + -25.899;
   1:  PR[GP1:91,2] = PR[GP1:90,2] + -16.037;
   1:L PR[91] R[100]mm/sec CNT100;
   1:  PR[GP1:91,1] = PR[GP1:90,1] + -24.399;
   1:  PR[GP1:91,2] = PR[GP1:90,2] + -17.210;
   1:L PR[91] R[100]mm/sec CNT100;
   1:  PR[GP1:91,1] = PR[GP1:90,1] + -21.126;
   1:  PR[GP1:91,2] = PR[GP1:90,2] + -19.637;
   1:L PR[91] R[100]mm/sec CNT100;
   1:  PR[GP1:91,1] = PR[GP1:90,1] + -19.060;
   1:  PR[GP1:91,2] = PR[GP1:90,2] + -20.536;
   1:L PR[91] R[100]mm/sec CNT100;
   1:  PR[GP1:91,1] = PR[GP1:90,1] + -15.535;
   1:  PR[GP1:91,2] = PR[GP1:90,2] + -21.957;
   1:L PR[91] R[100]mm/sec CNT100;
   1:  PR[GP1:91,1] = PR[GP1:90,1] + -12.948;
   1:  PR[GP1:91,2] = PR[GP1:90,2] + -22.368;
   1:L PR[91] R[100]mm/sec CNT100;
   1:  PR[GP1:91,1] = PR[GP1:90,1] + -9.506;
   1:  PR[GP1:91,2] = PR[GP1:90,2] + -22.814;
   1:L PR[91] R[100]mm/sec CNT100;
   1:  PR[GP1:91,1] = PR[GP1:90,1] + -6.457;
   1:  PR[GP1:91,2] = PR[GP1:90,2] + -22.513;
   1:L PR[91] R[100]mm/sec CNT100;
   1:  PR[GP1:91,1] = PR[GP1:90,1] + -3.417;
   1:  PR[GP1:91,2] = PR[GP1:90,2] + -22.124;
   1:L PR[91] R[100]mm/sec CNT100;
   1:  PR[GP1:91,1] = PR[GP1:90,1] + -0.720;
   1:  PR[GP1:91,2] = PR[GP1:90,2] + -21.186;
   1:L PR[91] R[100]mm/sec CNT100;
   1:  PR[GP1:91,1] = PR[GP1:90,1] + -0.418;
   1:  PR[GP1:91,2] = PR[GP1:90,2] + -21.193;
   1:L PR[91] R[100]mm/sec CNT100;
   1:  PR[GP1:91,1] = PR[GP1:90,1] + 0.738;
   1:  PR[GP1:91,2] = PR[GP1:90,2] + -21.048;
   1:L PR[91] R[100]mm/sec CNT100;
   1:  PR[GP1:91,1] = PR[GP1:90,1] + 1.236;
   1:  PR[GP1:91,2] = PR[GP1:90,2] + -21.315;
   1:L PR[91] R[100]mm/sec CNT100;
   1:  PR[GP1:91,1] = PR[GP1:90,1] + 2.676;
   1:  PR[GP1:91,2] = PR[GP1:90,2] + -21.832;
   1:L PR[91] R[100]mm/sec CNT100;
   1:  PR[GP1:91,1] = PR[GP1:90,1] + 3.246;
   1:  PR[GP1:91,2] = PR[GP1:90,2] + -22.022;
   1:L PR[91] R[100]mm/sec CNT100;
   1:  PR[GP1:91,1] = PR[GP1:90,1] + 6.021;
   1:  PR[GP1:91,2] = PR[GP1:90,2] + -22.381;
   1:L PR[91] R[100]mm/sec CNT100;
   1:  PR[GP1:91,1] = PR[GP1:90,1] + 6.672;
   1:  PR[GP1:91,2] = PR[GP1:90,2] + -22.519;
   1:L PR[91] R[100]mm/sec CNT100;
   1:  PR[GP1:91,1] = PR[GP1:90,1] + 9.662;
   1:  PR[GP1:91,2] = PR[GP1:90,2] + -22.814;
   1:L PR[91] R[100]mm/sec CNT100;
   1:  PR[GP1:91,1] = PR[GP1:90,1] + 13.104;
   1:  PR[GP1:91,2] = PR[GP1:90,2] + -22.368;
   1:L PR[91] R[100]mm/sec CNT100;
   1:  PR[GP1:91,1] = PR[GP1:90,1] + 15.691;
   1:  PR[GP1:91,2] = PR[GP1:90,2] + -21.957;
   1:L PR[91] R[100]mm/sec CNT100;
   1:  PR[GP1:91,1] = PR[GP1:90,1] + 19.217;
   1:  PR[GP1:91,2] = PR[GP1:90,2] + -20.537;
   1:L PR[91] R[100]mm/sec CNT100;
   1:  PR[GP1:91,1] = PR[GP1:90,1] + 21.282;
   1:  PR[GP1:91,2] = PR[GP1:90,2] + -19.638;
   1:L PR[91] R[100]mm/sec CNT100;
   1:  PR[GP1:91,1] = PR[GP1:90,1] + 24.555;
   1:  PR[GP1:91,2] = PR[GP1:90,2] + -17.212;
   1:L PR[91] R[100]mm/sec CNT100;
   1:  PR[GP1:91,1] = PR[GP1:90,1] + 26.055;
   1:  PR[GP1:91,2] = PR[GP1:90,2] + -16.038;
   1:L PR[91] R[100]mm/sec CNT100;
   1:  PR[GP1:91,1] = PR[GP1:90,1] + 28.717;
   1:  PR[GP1:91,2] = PR[GP1:90,2] + -12.675;
   1:L PR[91] R[100]mm/sec CNT100;
   1:  PR[GP1:91,1] = PR[GP1:90,1] + 29.704;
   1:  PR[GP1:91,2] = PR[GP1:90,2] + -11.378;
   1:L PR[91] R[100]mm/sec CNT100;
   1:  PR[GP1:91,1] = PR[GP1:90,1] + 31.440;
   1:  PR[GP1:91,2] = PR[GP1:90,2] + -7.385;
   1:L PR[91] R[100]mm/sec CNT100;
   1:  PR[GP1:91,1] = PR[GP1:90,1] + 31.985;
   1:  PR[GP1:91,2] = PR[GP1:90,2] + -6.071;
   1:L PR[91] R[100]mm/sec CNT100;
   1:  PR[GP1:91,1] = PR[GP1:90,1] + 32.586;
   1:  PR[GP1:91,2] = PR[GP1:90,2] + -1.630;
   1:L PR[91] R[100]mm/sec CNT100;
   1:  PR[GP1:91,1] = PR[GP1:90,1] + 32.714;
   1:  PR[GP1:91,2] = PR[GP1:90,2] + -0.338;
   1:L PR[91] R[100]mm/sec CNT100;
   1:  PR[GP1:91,1] = PR[GP1:90,1] + 32.286;
   1:  PR[GP1:91,2] = PR[GP1:90,2] + 2.809;
   1:L PR[91] R[100]mm/sec CNT100;
   1:  PR[GP1:91,1] = PR[GP1:90,1] + 32.165;
   1:  PR[GP1:91,2] = PR[GP1:90,2] + 4.085;
   1:L PR[91] R[100]mm/sec CNT100;
   1:  PR[GP1:91,1] = PR[GP1:90,1] + 31.986;
   1:  PR[GP1:91,2] = PR[GP1:90,2] + 5.443;
   1:L PR[91] R[100]mm/sec CNT100;
   1:  PR[GP1:91,1] = PR[GP1:90,1] + 31.443;
   1:  PR[GP1:91,2] = PR[GP1:90,2] + 6.753;
   1:L PR[91] R[100]mm/sec CNT100;
   1:  PR[GP1:91,1] = PR[GP1:90,1] + 29.711;
   1:  PR[GP1:91,2] = PR[GP1:90,2] + 10.742;
   1:L PR[91] R[100]mm/sec CNT100;
   1:  PR[GP1:91,1] = PR[GP1:90,1] + 28.726;
   1:  PR[GP1:91,2] = PR[GP1:90,2] + 12.038;
   1:L PR[91] R[100]mm/sec CNT100;
   1:  PR[GP1:91,1] = PR[GP1:90,1] + 26.070;
   1:  PR[GP1:91,2] = PR[GP1:90,2] + 15.400;
   1:L PR[91] R[100]mm/sec CNT100;
   1:  PR[GP1:91,1] = PR[GP1:90,1] + 24.573;
   1:  PR[GP1:91,2] = PR[GP1:90,2] + 16.573;
   1:L PR[91] R[100]mm/sec CNT100;
   1:  PR[GP1:91,1] = PR[GP1:90,1] + 21.306;
   1:  PR[GP1:91,2] = PR[GP1:90,2] + 19.001;
   1:L PR[91] R[100]mm/sec CNT100;
   1:  PR[GP1:91,1] = PR[GP1:90,1] + 19.245;
   1:  PR[GP1:91,2] = PR[GP1:90,2] + 19.900;
   1:L PR[91] R[100]mm/sec CNT100;
   1:  PR[GP1:91,1] = PR[GP1:90,1] + 15.724;
   1:  PR[GP1:91,2] = PR[GP1:90,2] + 21.324;
   1:L PR[91] R[100]mm/sec CNT100;
   1:  PR[GP1:91,1] = PR[GP1:90,1] + 13.142;
   1:  PR[GP1:91,2] = PR[GP1:90,2] + 21.738;
   1:L PR[91] R[100]mm/sec CNT100;
   1:  PR[GP1:91,1] = PR[GP1:90,1] + 9.702;
   1:  PR[GP1:91,2] = PR[GP1:90,2] + 22.190;
   1:L PR[91] R[100]mm/sec CNT100;
   1:  PR[GP1:91,1] = PR[GP1:90,1] + 6.685;
   1:  PR[GP1:91,2] = PR[GP1:90,2] + 21.899;
   1:L PR[91] R[100]mm/sec CNT100;
   1:  PR[GP1:91,1] = PR[GP1:90,1] + 3.607;
   1:  PR[GP1:91,2] = PR[GP1:90,2] + 21.511;
   1:L PR[91] R[100]mm/sec CNT100;
   1:  PR[GP1:91,1] = PR[GP1:90,1] + 2.703;
   1:  PR[GP1:91,2] = PR[GP1:90,2] + 21.216;
   1:L PR[91] R[100]mm/sec CNT100;
   1:  PR[GP1:91,1] = PR[GP1:90,1] + 1.200;
   1:  PR[GP1:91,2] = PR[GP1:90,2] + 20.665;
   1:L PR[91] R[100]mm/sec CNT100;
   1:  PR[GP1:91,1] = PR[GP1:90,1] + 0.667;
   1:  PR[GP1:91,2] = PR[GP1:90,2] + 20.418;
   1:L PR[91] R[100]mm/sec CNT100;
   1:  ! -- Layer/Ebene 82 -- !;
   1:  PR[91] = PR[90];
   1:  PR[GP1:91,1] = PR[GP1:90,1] + -0.077;
   1:  PR[GP1:91,2] = PR[GP1:90,2] + 20.737;
   1:  PR[GP1:91,3] = PR[GP1:90,3] + 50.325;
   1:L PR[91] R[100]mm/sec CNT100;
   1:  PR[GP1:91,1] = PR[GP1:90,1] + -0.719;
   1:  PR[GP1:91,2] = PR[GP1:90,2] + 20.727;
   1:L PR[91] R[100]mm/sec CNT100;
   1:  PR[GP1:91,1] = PR[GP1:90,1] + -2.646;
   1:  PR[GP1:91,2] = PR[GP1:90,2] + 21.430;
   1:L PR[91] R[100]mm/sec CNT100;
   1:  PR[GP1:91,1] = PR[GP1:90,1] + -3.230;
   1:  PR[GP1:91,2] = PR[GP1:90,2] + 21.617;
   1:L PR[91] R[100]mm/sec CNT100;
   1:  PR[GP1:91,1] = PR[GP1:90,1] + -6.066;
   1:  PR[GP1:91,2] = PR[GP1:90,2] + 21.973;
   1:L PR[91] R[100]mm/sec CNT100;
   1:  PR[GP1:91,1] = PR[GP1:90,1] + -9.347;
   1:  PR[GP1:91,2] = PR[GP1:90,2] + 22.289;
   1:L PR[91] R[100]mm/sec CNT100;
   1:  PR[GP1:91,1] = PR[GP1:90,1] + -12.537;
   1:  PR[GP1:91,2] = PR[GP1:90,2] + 21.870;
   1:L PR[91] R[100]mm/sec CNT100;
   1:  PR[GP1:91,1] = PR[GP1:90,1] + -15.384;
   1:  PR[GP1:91,2] = PR[GP1:90,2] + 21.414;
   1:L PR[91] R[100]mm/sec CNT100;
   1:  PR[GP1:91,1] = PR[GP1:90,1] + -18.664;
   1:  PR[GP1:91,2] = PR[GP1:90,2] + 20.086;
   1:L PR[91] R[100]mm/sec CNT100;
   1:  PR[GP1:91,1] = PR[GP1:90,1] + -20.978;
   1:  PR[GP1:91,2] = PR[GP1:90,2] + 19.076;
   1:L PR[91] R[100]mm/sec CNT100;
   1:  PR[GP1:91,1] = PR[GP1:90,1] + -24.034;
   1:  PR[GP1:91,2] = PR[GP1:90,2] + 16.805;
   1:L PR[91] R[100]mm/sec CNT100;
   1:  PR[GP1:91,1] = PR[GP1:90,1] + -25.752;
   1:  PR[GP1:91,2] = PR[GP1:90,2] + 15.459;
   1:L PR[91] R[100]mm/sec CNT100;
   1:  PR[GP1:91,1] = PR[GP1:90,1] + -28.245;
   1:  PR[GP1:91,2] = PR[GP1:90,2] + 12.310;
   1:L PR[91] R[100]mm/sec CNT100;
   1:  PR[GP1:91,1] = PR[GP1:90,1] + -29.399;
   1:  PR[GP1:91,2] = PR[GP1:90,2] + 10.791;
   1:L PR[91] R[100]mm/sec CNT100;
   1:  PR[GP1:91,1] = PR[GP1:90,1] + -31.027;
   1:  PR[GP1:91,2] = PR[GP1:90,2] + 7.025;
   1:L PR[91] R[100]mm/sec CNT100;
   1:  PR[GP1:91,1] = PR[GP1:90,1] + -31.680;
   1:  PR[GP1:91,2] = PR[GP1:90,2] + 5.448;
   1:L PR[91] R[100]mm/sec CNT100;
   1:  PR[GP1:91,1] = PR[GP1:90,1] + -32.244;
   1:  PR[GP1:91,2] = PR[GP1:90,2] + 1.285;
   1:L PR[91] R[100]mm/sec CNT100;
   1:  PR[GP1:91,1] = PR[GP1:90,1] + -32.399;
   1:  PR[GP1:91,2] = PR[GP1:90,2] + -0.285;
   1:L PR[91] R[100]mm/sec CNT100;
   1:  PR[GP1:91,1] = PR[GP1:90,1] + -32.035;
   1:  PR[GP1:91,2] = PR[GP1:90,2] + -2.954;
   1:L PR[91] R[100]mm/sec CNT100;
   1:  PR[GP1:91,1] = PR[GP1:90,1] + -31.892;
   1:  PR[GP1:91,2] = PR[GP1:90,2] + -4.449;
   1:L PR[91] R[100]mm/sec CNT100;
   1:  PR[GP1:91,1] = PR[GP1:90,1] + -31.677;
   1:  PR[GP1:91,2] = PR[GP1:90,2] + -6.081;
   1:L PR[91] R[100]mm/sec CNT100;
   1:  PR[GP1:91,1] = PR[GP1:90,1] + -31.024;
   1:  PR[GP1:91,2] = PR[GP1:90,2] + -7.656;
   1:L PR[91] R[100]mm/sec CNT100;
   1:  PR[GP1:91,1] = PR[GP1:90,1] + -29.392;
   1:  PR[GP1:91,2] = PR[GP1:90,2] + -11.427;
   1:L PR[91] R[100]mm/sec CNT100;
   1:  PR[GP1:91,1] = PR[GP1:90,1] + -28.235;
   1:  PR[GP1:91,2] = PR[GP1:90,2] + -12.947;
   1:L PR[91] R[100]mm/sec CNT100;
   1:  PR[GP1:91,1] = PR[GP1:90,1] + -25.737;
   1:  PR[GP1:91,2] = PR[GP1:90,2] + -16.097;
   1:L PR[91] R[100]mm/sec CNT100;
   1:  PR[GP1:91,1] = PR[GP1:90,1] + -24.016;
   1:  PR[GP1:91,2] = PR[GP1:90,2] + -17.444;
   1:L PR[91] R[100]mm/sec CNT100;
   1:  PR[GP1:91,1] = PR[GP1:90,1] + -20.954;
   1:  PR[GP1:91,2] = PR[GP1:90,2] + -19.714;
   1:L PR[91] R[100]mm/sec CNT100;
   1:  PR[GP1:91,1] = PR[GP1:90,1] + -18.636;
   1:  PR[GP1:91,2] = PR[GP1:90,2] + -20.723;
   1:L PR[91] R[100]mm/sec CNT100;
   1:  PR[GP1:91,1] = PR[GP1:90,1] + -15.351;
   1:  PR[GP1:91,2] = PR[GP1:90,2] + -22.047;
   1:L PR[91] R[100]mm/sec CNT100;
   1:  PR[GP1:91,1] = PR[GP1:90,1] + -12.499;
   1:  PR[GP1:91,2] = PR[GP1:90,2] + -22.500;
   1:L PR[91] R[100]mm/sec CNT100;
   1:  PR[GP1:91,1] = PR[GP1:90,1] + -9.307;
   1:  PR[GP1:91,2] = PR[GP1:90,2] + -22.914;
   1:L PR[91] R[100]mm/sec CNT100;
   1:  PR[GP1:91,1] = PR[GP1:90,1] + -5.992;
   1:  PR[GP1:91,2] = PR[GP1:90,2] + -22.586;
   1:L PR[91] R[100]mm/sec CNT100;
   1:  PR[GP1:91,1] = PR[GP1:90,1] + -3.179;
   1:  PR[GP1:91,2] = PR[GP1:90,2] + -22.227;
   1:L PR[91] R[100]mm/sec CNT100;
   1:  PR[GP1:91,1] = PR[GP1:90,1] + -2.983;
   1:  PR[GP1:91,2] = PR[GP1:90,2] + -22.165;
   1:L PR[91] R[100]mm/sec CNT100;
   1:  PR[GP1:91,1] = PR[GP1:90,1] + -0.707;
   1:  PR[GP1:91,2] = PR[GP1:90,2] + -21.363;
   1:L PR[91] R[100]mm/sec CNT100;
   1:  PR[GP1:91,1] = PR[GP1:90,1] + -0.258;
   1:  PR[GP1:91,2] = PR[GP1:90,2] + -21.372;
   1:L PR[91] R[100]mm/sec CNT100;
   1:  PR[GP1:91,1] = PR[GP1:90,1] + 0.756;
   1:  PR[GP1:91,2] = PR[GP1:90,2] + -21.245;
   1:L PR[91] R[100]mm/sec CNT100;
   1:  PR[GP1:91,1] = PR[GP1:90,1] + 1.220;
   1:  PR[GP1:91,2] = PR[GP1:90,2] + -21.494;
   1:L PR[91] R[100]mm/sec CNT100;
   1:  PR[GP1:91,1] = PR[GP1:90,1] + 2.385;
   1:  PR[GP1:91,2] = PR[GP1:90,2] + -21.913;
   1:L PR[91] R[100]mm/sec CNT100;
   1:  PR[GP1:91,1] = PR[GP1:90,1] + 3.007;
   1:  PR[GP1:91,2] = PR[GP1:90,2] + -22.120;
   1:L PR[91] R[100]mm/sec CNT100;
   1:  PR[GP1:91,1] = PR[GP1:90,1] + 5.501;
   1:  PR[GP1:91,2] = PR[GP1:90,2] + -22.443;
   1:L PR[91] R[100]mm/sec CNT100;
   1:  PR[GP1:91,1] = PR[GP1:90,1] + 6.207;
   1:  PR[GP1:91,2] = PR[GP1:90,2] + -22.592;
   1:L PR[91] R[100]mm/sec CNT100;
   1:  PR[GP1:91,1] = PR[GP1:90,1] + 9.463;
   1:  PR[GP1:91,2] = PR[GP1:90,2] + -22.914;
   1:L PR[91] R[100]mm/sec CNT100;
   1:  PR[GP1:91,1] = PR[GP1:90,1] + 12.655;
   1:  PR[GP1:91,2] = PR[GP1:90,2] + -22.500;
   1:L PR[91] R[100]mm/sec CNT100;
   1:  PR[GP1:91,1] = PR[GP1:90,1] + 15.507;
   1:  PR[GP1:91,2] = PR[GP1:90,2] + -22.047;
   1:L PR[91] R[100]mm/sec CNT100;
   1:  PR[GP1:91,1] = PR[GP1:90,1] + 18.793;
   1:  PR[GP1:91,2] = PR[GP1:90,2] + -20.723;
   1:L PR[91] R[100]mm/sec CNT100;
   1:  PR[GP1:91,1] = PR[GP1:90,1] + 21.110;
   1:  PR[GP1:91,2] = PR[GP1:90,2] + -19.715;
   1:L PR[91] R[100]mm/sec CNT100;
   1:  PR[GP1:91,1] = PR[GP1:90,1] + 24.172;
   1:  PR[GP1:91,2] = PR[GP1:90,2] + -17.445;
   1:L PR[91] R[100]mm/sec CNT100;
   1:  PR[GP1:91,1] = PR[GP1:90,1] + 25.893;
   1:  PR[GP1:91,2] = PR[GP1:90,2] + -16.099;
   1:L PR[91] R[100]mm/sec CNT100;
   1:  PR[GP1:91,1] = PR[GP1:90,1] + 28.391;
   1:  PR[GP1:91,2] = PR[GP1:90,2] + -12.943;
   1:L PR[91] R[100]mm/sec CNT100;
   1:  PR[GP1:91,1] = PR[GP1:90,1] + 29.549;
   1:  PR[GP1:91,2] = PR[GP1:90,2] + -11.420;
   1:L PR[91] R[100]mm/sec CNT100;
   1:  PR[GP1:91,1] = PR[GP1:90,1] + 31.181;
   1:  PR[GP1:91,2] = PR[GP1:90,2] + -7.666;
   1:L PR[91] R[100]mm/sec CNT100;
   1:  PR[GP1:91,1] = PR[GP1:90,1] + 31.835;
   1:  PR[GP1:91,2] = PR[GP1:90,2] + -6.091;
   1:L PR[91] R[100]mm/sec CNT100;
   1:  PR[GP1:91,1] = PR[GP1:90,1] + 32.400;
   1:  PR[GP1:91,2] = PR[GP1:90,2] + -1.912;
   1:L PR[91] R[100]mm/sec CNT100;
   1:  PR[GP1:91,1] = PR[GP1:90,1] + 32.556;
   1:  PR[GP1:91,2] = PR[GP1:90,2] + -0.338;
   1:L PR[91] R[100]mm/sec CNT100;
   1:  PR[GP1:91,1] = PR[GP1:90,1] + 32.193;
   1:  PR[GP1:91,2] = PR[GP1:90,2] + 2.336;
   1:L PR[91] R[100]mm/sec CNT100;
   1:  PR[GP1:91,1] = PR[GP1:90,1] + 32.050;
   1:  PR[GP1:91,2] = PR[GP1:90,2] + 3.832;
   1:L PR[91] R[100]mm/sec CNT100;
   1:  PR[GP1:91,1] = PR[GP1:90,1] + 31.835;
   1:  PR[GP1:91,2] = PR[GP1:90,2] + 5.463;
   1:L PR[91] R[100]mm/sec CNT100;
   1:  PR[GP1:91,1] = PR[GP1:90,1] + 31.184;
   1:  PR[GP1:91,2] = PR[GP1:90,2] + 7.034;
   1:L PR[91] R[100]mm/sec CNT100;
   1:  PR[GP1:91,1] = PR[GP1:90,1] + 29.556;
   1:  PR[GP1:91,2] = PR[GP1:90,2] + 10.785;
   1:L PR[91] R[100]mm/sec CNT100;
   1:  PR[GP1:91,1] = PR[GP1:90,1] + 28.401;
   1:  PR[GP1:91,2] = PR[GP1:90,2] + 12.306;
   1:L PR[91] R[100]mm/sec CNT100;
   1:  PR[GP1:91,1] = PR[GP1:90,1] + 25.908;
   1:  PR[GP1:91,2] = PR[GP1:90,2] + 15.461;
   1:L PR[91] R[100]mm/sec CNT100;
   1:  PR[GP1:91,1] = PR[GP1:90,1] + 24.191;
   1:  PR[GP1:91,2] = PR[GP1:90,2] + 16.806;
   1:L PR[91] R[100]mm/sec CNT100;
   1:  PR[GP1:91,1] = PR[GP1:90,1] + 21.134;
   1:  PR[GP1:91,2] = PR[GP1:90,2] + 19.078;
   1:L PR[91] R[100]mm/sec CNT100;
   1:  PR[GP1:91,1] = PR[GP1:90,1] + 18.821;
   1:  PR[GP1:91,2] = PR[GP1:90,2] + 20.087;
   1:L PR[91] R[100]mm/sec CNT100;
   1:  PR[GP1:91,1] = PR[GP1:90,1] + 15.540;
   1:  PR[GP1:91,2] = PR[GP1:90,2] + 21.414;
   1:L PR[91] R[100]mm/sec CNT100;
   1:  PR[GP1:91,1] = PR[GP1:90,1] + 12.693;
   1:  PR[GP1:91,2] = PR[GP1:90,2] + 21.870;
   1:L PR[91] R[100]mm/sec CNT100;
   1:  PR[GP1:91,1] = PR[GP1:90,1] + 9.503;
   1:  PR[GP1:91,2] = PR[GP1:90,2] + 22.289;
   1:L PR[91] R[100]mm/sec CNT100;
   1:  PR[GP1:91,1] = PR[GP1:90,1] + 6.223;
   1:  PR[GP1:91,2] = PR[GP1:90,2] + 21.973;
   1:L PR[91] R[100]mm/sec CNT100;
   1:  PR[GP1:91,1] = PR[GP1:90,1] + 3.391;
   1:  PR[GP1:91,2] = PR[GP1:90,2] + 21.616;
   1:L PR[91] R[100]mm/sec CNT100;
   1:  PR[GP1:91,1] = PR[GP1:90,1] + 2.410;
   1:  PR[GP1:91,2] = PR[GP1:90,2] + 21.296;
   1:L PR[91] R[100]mm/sec CNT100;
   1:  PR[GP1:91,1] = PR[GP1:90,1] + 1.185;
   1:  PR[GP1:91,2] = PR[GP1:90,2] + 20.847;
   1:L PR[91] R[100]mm/sec CNT100;
   1:  PR[GP1:91,1] = PR[GP1:90,1] + 0.684;
   1:  PR[GP1:91,2] = PR[GP1:90,2] + 20.615;
   1:L PR[91] R[100]mm/sec CNT100;
   1:  ! -- Layer/Ebene 83 -- !;
   1:  PR[91] = PR[90];
   1:  PR[GP1:91,1] = PR[GP1:90,1] + 0.036;
   1:  PR[GP1:91,2] = PR[GP1:90,2] + 20.919;
   1:  PR[GP1:91,3] = PR[GP1:90,3] + 50.935;
   1:L PR[91] R[100]mm/sec CNT100;
   1:  PR[GP1:91,1] = PR[GP1:90,1] + -0.703;
   1:  PR[GP1:91,2] = PR[GP1:90,2] + 20.908;
   1:L PR[91] R[100]mm/sec CNT100;
   1:  PR[GP1:91,1] = PR[GP1:90,1] + -2.379;
   1:  PR[GP1:91,2] = PR[GP1:90,2] + 21.519;
   1:L PR[91] R[100]mm/sec CNT100;
   1:  PR[GP1:91,1] = PR[GP1:90,1] + -3.014;
   1:  PR[GP1:91,2] = PR[GP1:90,2] + 21.722;
   1:L PR[91] R[100]mm/sec CNT100;
   1:  PR[GP1:91,1] = PR[GP1:90,1] + -5.604;
   1:  PR[GP1:91,2] = PR[GP1:90,2] + 22.047;
   1:L PR[91] R[100]mm/sec CNT100;
   1:  PR[GP1:91,1] = PR[GP1:90,1] + -9.148;
   1:  PR[GP1:91,2] = PR[GP1:90,2] + 22.389;
   1:L PR[91] R[100]mm/sec CNT100;
   1:  PR[GP1:91,1] = PR[GP1:90,1] + -12.088;
   1:  PR[GP1:91,2] = PR[GP1:90,2] + 22.003;
   1:L PR[91] R[100]mm/sec CNT100;
   1:  PR[GP1:91,1] = PR[GP1:90,1] + -15.199;
   1:  PR[GP1:91,2] = PR[GP1:90,2] + 21.504;
   1:L PR[91] R[100]mm/sec CNT100;
   1:  PR[GP1:91,1] = PR[GP1:90,1] + -18.240;
   1:  PR[GP1:91,2] = PR[GP1:90,2] + 20.273;
   1:L PR[91] R[100]mm/sec CNT100;
   1:  PR[GP1:91,1] = PR[GP1:90,1] + -20.806;
   1:  PR[GP1:91,2] = PR[GP1:90,2] + 19.154;
   1:L PR[91] R[100]mm/sec CNT100;
   1:  PR[GP1:91,1] = PR[GP1:90,1] + -23.652;
   1:  PR[GP1:91,2] = PR[GP1:90,2] + 17.038;
   1:L PR[91] R[100]mm/sec CNT100;
   1:  PR[GP1:91,1] = PR[GP1:90,1] + -25.590;
   1:  PR[GP1:91,2] = PR[GP1:90,2] + 15.520;
   1:L PR[91] R[100]mm/sec CNT100;
   1:  PR[GP1:91,1] = PR[GP1:90,1] + -27.919;
   1:  PR[GP1:91,2] = PR[GP1:90,2] + 12.578;
   1:L PR[91] R[100]mm/sec CNT100;
   1:  PR[GP1:91,1] = PR[GP1:90,1] + -29.244;
   1:  PR[GP1:91,2] = PR[GP1:90,2] + 10.833;
   1:L PR[91] R[100]mm/sec CNT100;
   1:  PR[GP1:91,1] = PR[GP1:90,1] + -30.769;
   1:  PR[GP1:91,2] = PR[GP1:90,2] + 7.305;
   1:L PR[91] R[100]mm/sec CNT100;
   1:  PR[GP1:91,1] = PR[GP1:90,1] + -31.529;
   1:  PR[GP1:91,2] = PR[GP1:90,2] + 5.469;
   1:L PR[91] R[100]mm/sec CNT100;
   1:  PR[GP1:91,1] = PR[GP1:90,1] + -32.058;
   1:  PR[GP1:91,2] = PR[GP1:90,2] + 1.566;
   1:L PR[91] R[100]mm/sec CNT100;
   1:  PR[GP1:91,1] = PR[GP1:90,1] + -32.242;
   1:  PR[GP1:91,2] = PR[GP1:90,2] + -0.285;
   1:L PR[91] R[100]mm/sec CNT100;
   1:  PR[GP1:91,1] = PR[GP1:90,1] + -31.942;
   1:  PR[GP1:91,2] = PR[GP1:90,2] + -2.482;
   1:L PR[91] R[100]mm/sec CNT100;
   1:  PR[GP1:91,1] = PR[GP1:90,1] + -31.778;
   1:  PR[GP1:91,2] = PR[GP1:90,2] + -4.197;
   1:L PR[91] R[100]mm/sec CNT100;
   1:  PR[GP1:91,1] = PR[GP1:90,1] + -31.526;
   1:  PR[GP1:91,2] = PR[GP1:90,2] + -6.102;
   1:L PR[91] R[100]mm/sec CNT100;
   1:  PR[GP1:91,1] = PR[GP1:90,1] + -30.766;
   1:  PR[GP1:91,2] = PR[GP1:90,2] + -7.938;
   1:L PR[91] R[100]mm/sec CNT100;
   1:  PR[GP1:91,1] = PR[GP1:90,1] + -29.237;
   1:  PR[GP1:91,2] = PR[GP1:90,2] + -11.469;
   1:L PR[91] R[100]mm/sec CNT100;
   1:  PR[GP1:91,1] = PR[GP1:90,1] + -27.909;
   1:  PR[GP1:91,2] = PR[GP1:90,2] + -13.215;
   1:L PR[91] R[100]mm/sec CNT100;
   1:  PR[GP1:91,1] = PR[GP1:90,1] + -25.575;
   1:  PR[GP1:91,2] = PR[GP1:90,2] + -16.158;
   1:L PR[91] R[100]mm/sec CNT100;
   1:  PR[GP1:91,1] = PR[GP1:90,1] + -23.633;
   1:  PR[GP1:91,2] = PR[GP1:90,2] + -17.677;
   1:L PR[91] R[100]mm/sec CNT100;
   1:  PR[GP1:91,1] = PR[GP1:90,1] + -20.782;
   1:  PR[GP1:91,2] = PR[GP1:90,2] + -19.791;
   1:L PR[91] R[100]mm/sec CNT100;
   1:  PR[GP1:91,1] = PR[GP1:90,1] + -18.211;
   1:  PR[GP1:91,2] = PR[GP1:90,2] + -20.909;
   1:L PR[91] R[100]mm/sec CNT100;
   1:  PR[GP1:91,1] = PR[GP1:90,1] + -15.166;
   1:  PR[GP1:91,2] = PR[GP1:90,2] + -22.137;
   1:L PR[91] R[100]mm/sec CNT100;
   1:  PR[GP1:91,1] = PR[GP1:90,1] + -12.050;
   1:  PR[GP1:91,2] = PR[GP1:90,2] + -22.632;
   1:L PR[91] R[100]mm/sec CNT100;
   1:  PR[GP1:91,1] = PR[GP1:90,1] + -9.108;
   1:  PR[GP1:91,2] = PR[GP1:90,2] + -23.013;
   1:L PR[91] R[100]mm/sec CNT100;
   1:  PR[GP1:91,1] = PR[GP1:90,1] + -5.527;
   1:  PR[GP1:91,2] = PR[GP1:90,2] + -22.659;
   1:L PR[91] R[100]mm/sec CNT100;
   1:  PR[GP1:91,1] = PR[GP1:90,1] + -2.963;
   1:  PR[GP1:91,2] = PR[GP1:90,2] + -22.332;
   1:L PR[91] R[100]mm/sec CNT100;
